LIN {X 0,Y 381.676,Z 552.93,A -85,B 0,C 180,E1 -11968.947,E2 -11968.947} C_VEL
LIN {X 0,Y 381.658,Z 553.223,A -85,B 0,C 180,E1 -11970.002,E2 -11970.002} C_VEL
LIN {X 0,Y 381.677,Z 553.115,A -85,B 0,C 180,E1 -11971.057,E2 -11971.057} C_VEL
LIN {X 0,Y 381.64,Z 552.556,A -85,B 0,C 180,E1 -11972.113,E2 -11972.113} C_VEL
LIN {X 0,Y 381.647,Z 550.205,A -85,B 0,C 180,E1 -11974.226,E2 -11974.226} C_VEL
LIN {X 0,Y 381.694,Z 546.609,A -85,B 0,C 180,E1 -11976.126,E2 -11976.126} C_VEL
LIN {X 0,Y 381.966,Z 541.741,A -85,B 0,C 180,E1 -11977.934,E2 -11977.934} C_VEL
LIN {X 0,Y 382.432,Z 535.151,A -85,B 0,C 180,E1 -11979.789,E2 -11979.789} C_VEL
LIN {X 0,Y 382.983,Z 527.932,A -85,B 0,C 180,E1 -11981.379,E2 -11981.379} C_VEL
LIN {X 0,Y 383.876,Z 518.998,A -85,B 0,C 180,E1 -11982.962,E2 -11982.962} C_VEL
LIN {X 0,Y 384.66,Z 509.425,A -85,B 0,C 180,E1 -11984.335,E2 -11984.335} C_VEL
LIN {X 0,Y 385.769,Z 498.433,A -85,B 0,C 180,E1 -11985.59,E2 -11985.59} C_VEL
LIN {X 0,Y 386.845,Z 487.015,A -85,B 0,C 180,E1 -11986.629,E2 -11986.629} C_VEL
LIN {X 0,Y 387.515,Z 477.015,A -85,B 0,C 180,E1 -11987.357,E2 -11987.357} C_VEL
LIN {X 0,Y 386.584,Z 463.507,A -85,B 0,C 180,E1 -11988.193,E2 -11988.193} C_VEL
LIN {X 0,Y 384.34,Z 449.997,A -85,B 0,C 180,E1 -11988.878,E2 -11988.878} C_VEL
LIN {X 0,Y 382.993,Z 443.041,A -85,B 0,C 180,E1 -11989.168,E2 -11989.168} C_VEL
LIN {X 0,Y 383.721,Z 433.258,A -85,B 0,C 180,E1 -11992.622,E2 -11992.622} C_VEL
LIN {X 0,Y 384.612,Z 423.855,A -85,B 0,C 180,E1 -11996.013,E2 -11996.013} C_VEL
LIN {X 0,Y 385.69,Z 414.532,A -85,B 0,C 180,E1 -11999.473,E2 -11999.473} C_VEL
LIN {X 0,Y 386.129,Z 410.031,A -85,B 0,C 180,E1 -12001.189,E2 -12001.189} C_VEL
LIN {X 0,Y 385.15,Z 403.611,A -85,B 0,C 180,E1 -12003.819,E2 -12003.819} C_VEL
LIN {X 0,Y 383.607,Z 395.835,A -85,B 0,C 180,E1 -12007.201,E2 -12007.201} C_VEL
LIN {X 0,Y 383.015,Z 392.777,A -85,B 0,C 180,E1 -12008.601,E2 -12008.601} C_VEL
LIN {X 0,Y 382.967,Z 392.783,A -85,B 0,C 180,E1 -12011.351,E2 -12011.351} C_VEL
LIN {X 0,Y 382.995,Z 392.777,A -85,B 0,C 180,E1 -12014.303,E2 -12014.303} C_VEL
LIN {X 0,Y 383.004,Z 392.776,A -85,B 0,C 180,E1 -12017.239,E2 -12017.239} C_VEL
LIN {X 0,Y 382.993,Z 392.777,A -85,B 0,C 180,E1 -12020.42,E2 -12020.42} C_VEL
LIN {X 0,Y 383.03,Z 392.774,A -85,B 0,C 180,E1 -12024.045,E2 -12024.045} C_VEL
LIN {X 0,Y 382.992,Z 392.778,A -85,B 0,C 180,E1 -12027.579,E2 -12027.579} C_VEL
LIN {X 0,Y 382.982,Z 392.779,A -85,B 0,C 180,E1 -12030.299,E2 -12030.299} C_VEL
LIN {X 0,Y 383.009,Z 392.775,A -85,B 0,C 180,E1 -12034.045,E2 -12034.045} C_VEL
LIN {X 0,Y 382.993,Z 392.778,A -85,B 0,C 180,E1 -12037.334,E2 -12037.334} C_VEL
LIN {X 0,Y 383.067,Z 392.771,A -85,B 0,C 180,E1 -12040.716,E2 -12040.716} C_VEL
LIN {X 0,Y 383.087,Z 392.771,A -85,B 0,C 180,E1 -12044.027,E2 -12044.027} C_VEL
LIN {X 0,Y 383.142,Z 392.763,A -85,B 0,C 180,E1 -12047.284,E2 -12047.284} C_VEL
LIN {X 0,Y 383.144,Z 392.76,A -85,B 0,C 180,E1 -12050.497,E2 -12050.497} C_VEL
LIN {X 0,Y 383.239,Z 392.75,A -85,B 0,C 180,E1 -12053.683,E2 -12053.683} C_VEL
LIN {X 0,Y 383.256,Z 392.948,A -85,B 0,C 180,E1 -12054.343,E2 -12054.343} C_VEL
LIN {X 0,Y 383.639,Z 397.881,A -85,B 0,C 180,E1 -12056.849,E2 -12056.849} C_VEL
LIN {X 0,Y 383.596,Z 403.09,A -85,B 0,C 180,E1 -12059.475,E2 -12059.475} C_VEL
LIN {X 0,Y 383.065,Z 411.611,A -85,B 0,C 180,E1 -12063.681,E2 -12063.681} C_VEL
LIN {X 0,Y 382.951,Z 417.902,A -85,B 0,C 180,E1 -12066.851,E2 -12066.851} C_VEL
LIN {X 0,Y 382.705,Z 424.252,A -85,B 0,C 180,E1 -12070.047,E2 -12070.047} C_VEL
LIN {X 0,Y 382.589,Z 427.474,A -85,B 0,C 180,E1 -12071.691,E2 -12071.691} C_VEL
LIN {X 0,Y 386.286,Z 441.807,A -85,B 0,C 180,E1 -12072.477,E2 -12072.477} C_VEL
LIN {X 0,Y 388.313,Z 452.899,A -85,B 0,C 180,E1 -12073.208,E2 -12073.208} C_VEL
LIN {X 0,Y 388.517,Z 456.626,A -85,B 0,C 180,E1 -12073.467,E2 -12073.467} C_VEL
LIN {X 0,Y 387.616,Z 468.027,A -85,B 0,C 180,E1 -12074.302,E2 -12074.302} C_VEL
LIN {X 0,Y 386.669,Z 479.198,A -85,B 0,C 180,E1 -12075.351,E2 -12075.351} C_VEL
LIN {X 0,Y 385.591,Z 490.485,A -85,B 0,C 180,E1 -12076.682,E2 -12076.682} C_VEL
LIN {X 0,Y 384.547,Z 500.254,A -85,B 0,C 180,E1 -12078.127,E2 -12078.127} C_VEL
LIN {X 0,Y 383.636,Z 509.359,A -85,B 0,C 180,E1 -12079.81,E2 -12079.81} C_VEL
LIN {X 0,Y 382.866,Z 516.695,A -85,B 0,C 180,E1 -12081.538,E2 -12081.538} C_VEL
LIN {X 0,Y 382.291,Z 522.218,A -85,B 0,C 180,E1 -12083.189,E2 -12083.189} C_VEL
LIN {X 0,Y 381.934,Z 526.91,A -85,B 0,C 180,E1 -12085.038,E2 -12085.038} C_VEL
LIN {X 0,Y 381.752,Z 529.124,A -85,B 0,C 180,E1 -12086.221,E2 -12086.221} C_VEL
LIN {X 0,Y 381.54,Z 531.322,A -85,B 0,C 180,E1 -12087.849,E2 -12087.849} C_VEL
LIN {X 0,Y 381.375,Z 532.743,A -85,B 0,C 180,E1 -12089.987,E2 -12089.987} C_VEL
LIN {X 0,Y 381.363,Z 532.498,A -85,B 0,C 180,E1 -12092.034,E2 -12092.034} C_VEL
LIN {X 0,Y 381.456,Z 530.872,A -85,B 0,C 180,E1 -12093.993,E2 -12093.993} C_VEL
LIN {X 0,Y 381.71,Z 527.886,A -85,B 0,C 180,E1 -12095.89,E2 -12095.89} C_VEL
LIN {X 0,Y 381.974,Z 523.67,A -85,B 0,C 180,E1 -12097.704,E2 -12097.704} C_VEL
LIN {X 0,Y 382.341,Z 518.193,A -85,B 0,C 180,E1 -12099.462,E2 -12099.462} C_VEL
LIN {X 0,Y 382.887,Z 511.233,A -85,B 0,C 180,E1 -12101.185,E2 -12101.185} C_VEL
LIN {X 0,Y 383.583,Z 502.634,A -85,B 0,C 180,E1 -12102.87,E2 -12102.87} C_VEL
LIN {X 0,Y 384.35,Z 493.592,A -85,B 0,C 180,E1 -12104.287,E2 -12104.287} C_VEL
LIN {X 0,Y 385.172,Z 483.42,A -85,B 0,C 180,E1 -12105.58,E2 -12105.58} C_VEL
LIN {X 0,Y 386.06,Z 472.137,A -85,B 0,C 180,E1 -12106.733,E2 -12106.733} C_VEL
LIN {X 0,Y 386.869,Z 460.044,A -85,B 0,C 180,E1 -12107.697,E2 -12107.697} C_VEL
LIN {X 0,Y 387.259,Z 452.848,A -85,B 0,C 180,E1 -12108.166,E2 -12108.166} C_VEL
LIN {X 0,Y 385.017,Z 440.265,A -85,B 0,C 180,E1 -12108.917,E2 -12108.917} C_VEL
LIN {X 0,Y 382.268,Z 426.607,A -85,B 0,C 180,E1 -12109.537,E2 -12109.537} C_VEL
LIN {X 0,Y 382.461,Z 419.18,A -85,B 0,C 180,E1 -12113.328,E2 -12113.328} C_VEL
LIN {X 0,Y 382.701,Z 412.84,A -85,B 0,C 180,E1 -12116.568,E2 -12116.568} C_VEL
LIN {X 0,Y 382.851,Z 406.873,A -85,B 0,C 180,E1 -12119.629,E2 -12119.629} C_VEL
LIN {X 0,Y 383.057,Z 399.753,A -85,B 0,C 180,E1 -12123.286,E2 -12123.286} C_VEL
LIN {X 0,Y 383.274,Z 394.063,A -85,B 0,C 180,E1 -12126.207,E2 -12126.207} C_VEL
LIN {X 0,Y 383.134,Z 392.763,A -85,B 0,C 180,E1 -12126.907,E2 -12126.907} C_VEL
LIN {X 0,Y 383.062,Z 392.772,A -85,B 0,C 180,E1 -12130.714,E2 -12130.714} C_VEL
LIN {X 0,Y 383.083,Z 392.767,A -85,B 0,C 180,E1 -12134.025,E2 -12134.025} C_VEL
LIN {X 0,Y 383.138,Z 392.76,A -85,B 0,C 180,E1 -12137.282,E2 -12137.282} C_VEL
LIN {X 0,Y 383.151,Z 392.758,A -85,B 0,C 180,E1 -12140.496,E2 -12140.496} C_VEL
LIN {X 0,Y 383.255,Z 392.748,A -85,B 0,C 180,E1 -12143.681,E2 -12143.681} C_VEL
LIN {X 0,Y 383.402,Z 392.882,A -85,B 0,C 180,E1 -12148.422,E2 -12148.422} C_VEL
LIN {X 0,Y 383.672,Z 395.201,A -85,B 0,C 180,E1 -12149.998,E2 -12149.998} C_VEL
LIN {X 0,Y 383.201,Z 400.099,A -85,B 0,C 180,E1 -12153.152,E2 -12153.152} C_VEL
LIN {X 0,Y 383.03,Z 405.091,A -85,B 0,C 180,E1 -12156.318,E2 -12156.318} C_VEL
LIN {X 0,Y 382.717,Z 410.229,A -85,B 0,C 180,E1 -12159.51,E2 -12159.51} C_VEL
LIN {X 0,Y 382.459,Z 416.09,A -85,B 0,C 180,E1 -12163.116,E2 -12163.116} C_VEL
LIN {X 0,Y 382.132,Z 422.772,A -85,B 0,C 180,E1 -12167.111,E2 -12167.111} C_VEL
LIN {X 0,Y 382.095,Z 423.941,A -85,B 0,C 180,E1 -12167.803,E2 -12167.803} C_VEL
LIN {X 0,Y 384.57,Z 436.385,A -85,B 0,C 180,E1 -12168.442,E2 -12168.442} C_VEL
LIN {X 0,Y 386.052,Z 446.599,A -85,B 0,C 180,E1 -12169.125,E2 -12169.125} C_VEL
LIN {X 0,Y 385.837,Z 451.459,A -85,B 0,C 180,E1 -12169.483,E2 -12169.483} C_VEL
LIN {X 0,Y 384.873,Z 456.639,A -85,B 0,C 180,E1 -12169.884,E2 -12169.884} C_VEL
LIN {X 0,Y 381.486,Z 464.749,A -85,B 0,C 180,E1 -12170.576,E2 -12170.576} C_VEL
LIN {X 0,Y 378.091,Z 472.32,A -85,B 0,C 180,E1 -12171.393,E2 -12171.393} C_VEL
LIN {X 0,Y 377.126,Z 476.647,A -85,B 0,C 180,E1 -12171.983,E2 -12171.983} C_VEL
LIN {X 0,Y 376.539,Z 483.312,A -85,B 0,C 180,E1 -12173.073,E2 -12173.073} C_VEL
LIN {X 0,Y 375.954,Z 490.705,A -85,B 0,C 180,E1 -12174.575,E2 -12174.575} C_VEL
LIN {X 0,Y 375.469,Z 496.349,A -85,B 0,C 180,E1 -12176.045,E2 -12176.045} C_VEL
LIN {X 0,Y 375.168,Z 500.199,A -85,B 0,C 180,E1 -12177.316,E2 -12177.316} C_VEL
LIN {X 0,Y 374.998,Z 502.515,A -85,B 0,C 180,E1 -12178.256,E2 -12178.256} C_VEL
LIN {X 0,Y 374.868,Z 504.313,A -85,B 0,C 180,E1 -12179.169,E2 -12179.169} C_VEL
LIN {X 0,Y 374.682,Z 506.2,A -85,B 0,C 180,E1 -12180.424,E2 -12180.424} C_VEL
LIN {X 0,Y 374.515,Z 507.759,A -85,B 0,C 180,E1 -12182.387,E2 -12182.387} C_VEL
LIN {X 0,Y 374.588,Z 507.67,A -85,B 0,C 180,E1 -12184.359,E2 -12184.359} C_VEL
LIN {X 0,Y 374.809,Z 506.038,A -85,B 0,C 180,E1 -12186.266,E2 -12186.266} C_VEL
LIN {X 0,Y 375.163,Z 502.8,A -85,B 0,C 180,E1 -12188.18,E2 -12188.18} C_VEL
LIN {X 0,Y 375.621,Z 498.336,A -85,B 0,C 180,E1 -12189.904,E2 -12189.904} C_VEL
LIN {X 0,Y 376.033,Z 493.712,A -85,B 0,C 180,E1 -12191.259,E2 -12191.259} C_VEL
LIN {X 0,Y 376.73,Z 486.408,A -85,B 0,C 180,E1 -12192.911,E2 -12192.911} C_VEL
LIN {X 0,Y 377.456,Z 478.658,A -85,B 0,C 180,E1 -12194.28,E2 -12194.28} C_VEL
LIN {X 0,Y 378.373,Z 469.354,A -85,B 0,C 180,E1 -12195.571,E2 -12195.571} C_VEL
LIN {X 0,Y 379.182,Z 459.767,A -85,B 0,C 180,E1 -12196.617,E2 -12196.617} C_VEL
LIN {X 0,Y 379.948,Z 448.957,A -85,B 0,C 180,E1 -12197.535,E2 -12197.535} C_VEL
LIN {X 0,Y 378.534,Z 439.629,A -85,B 0,C 180,E1 -12198.236,E2 -12198.236} C_VEL
LIN {X 0,Y 376.006,Z 428.04,A -85,B 0,C 180,E1 -12198.938,E2 -12198.938} C_VEL
LIN {X 0,Y 375.238,Z 424.84,A -85,B 0,C 180,E1 -12199.116,E2 -12199.116} C_VEL
LIN {X 0,Y 375.493,Z 419.416,A -85,B 0,C 180,E1 -12202.534,E2 -12202.534} C_VEL
LIN {X 0,Y 375.715,Z 414.233,A -85,B 0,C 180,E1 -12205.864,E2 -12205.864} C_VEL
LIN {X 0,Y 376.059,Z 408.313,A -85,B 0,C 180,E1 -12209.696,E2 -12209.696} C_VEL
LIN {X 0,Y 376.449,Z 402.826,A -85,B 0,C 180,E1 -12213.381,E2 -12213.381} C_VEL
LIN {X 0,Y 376.573,Z 398.851,A -85,B 0,C 180,E1 -12216.124,E2 -12216.124} C_VEL
LIN {X 0,Y 376.215,Z 394.642,A -85,B 0,C 180,E1 -12219.211,E2 -12219.211} C_VEL
LIN {X 0,Y 376.039,Z 393.648,A -85,B 0,C 180,E1 -12220.057,E2 -12220.057} C_VEL
LIN {X 0,Y 376.006,Z 393.654,A -85,B 0,C 180,E1 -12223.718,E2 -12223.718} C_VEL
LIN {X 0,Y 376.084,Z 393.64,A -85,B 0,C 180,E1 -12227.042,E2 -12227.042} C_VEL
LIN {X 0,Y 376.102,Z 393.638,A -85,B 0,C 180,E1 -12230.318,E2 -12230.318} C_VEL
LIN {X 0,Y 376.207,Z 393.625,A -85,B 0,C 180,E1 -12232.486,E2 -12232.486} C_VEL
LIN {X 0,Y 376.157,Z 393.631,A -85,B 0,C 180,E1 -12234.64,E2 -12234.64} C_VEL
LIN {X 0,Y 376.336,Z 393.608,A -85,B 0,C 180,E1 -12237.86,E2 -12237.86} C_VEL
LIN {X 0,Y 376.469,Z 393.592,A -85,B 0,C 180,E1 -12240,E2 -12240} C_VEL
LIN {X 0,Y 376.197,Z 393.624,A -85,B 0,C 180,E1 -12243.213,E2 -12243.213} C_VEL
LIN {X 0,Y 376.231,Z 393.616,A -85,B 0,C 180,E1 -12246.436,E2 -12246.436} C_VEL
LIN {X 0,Y 376.183,Z 393.627,A -85,B 0,C 180,E1 -12248.596,E2 -12248.596} C_VEL
LIN {X 0,Y 376.04,Z 393.643,A -85,B 0,C 180,E1 -12251.864,E2 -12251.864} C_VEL
LIN {X 0,Y 376.041,Z 393.642,A -85,B 0,C 180,E1 -12255.169,E2 -12255.169} C_VEL
LIN {X 0,Y 376.011,Z 393.643,A -85,B 0,C 180,E1 -12258.527,E2 -12258.527} C_VEL
LIN {X 0,Y 375.974,Z 393.65,A -85,B 0,C 180,E1 -12261.954,E2 -12261.954} C_VEL
LIN {X 0,Y 375.986,Z 393.651,A -85,B 0,C 180,E1 -12265.463,E2 -12265.463} C_VEL
LIN {X 0,Y 375.957,Z 393.653,A -85,B 0,C 180,E1 -12269.081,E2 -12269.081} C_VEL
LIN {X 0,Y 375.931,Z 393.655,A -85,B 0,C 180,E1 -12272.831,E2 -12272.831} C_VEL
LIN {X 0,Y 375.941,Z 393.657,A -85,B 0,C 180,E1 -12275.418,E2 -12275.418} C_VEL
LIN {X 0,Y 375.962,Z 393.656,A -85,B 0,C 180,E1 -12278.274,E2 -12278.274} C_VEL
LIN {X 0,Y 375.975,Z 393.654,A -85,B 0,C 180,E1 -12281.613,E2 -12281.613} C_VEL
LIN {X 0,Y 376.003,Z 393.647,A -85,B 0,C 180,E1 -12285.257,E2 -12285.257} C_VEL
LIN {X 0,Y 375.977,Z 393.652,A -85,B 0,C 180,E1 -12288.392,E2 -12288.392} C_VEL
LIN {X 0,Y 376.001,Z 393.84,A -85,B 0,C 180,E1 -12289.635,E2 -12289.635} C_VEL
LIN {X 0,Y 377.359,Z 400.688,A -85,B 0,C 180,E1 -12293.211,E2 -12293.211} C_VEL
LIN {X 0,Y 378.795,Z 407.795,A -85,B 0,C 180,E1 -12296.607,E2 -12296.607} C_VEL
LIN {X 0,Y 379.388,Z 412.708,A -85,B 0,C 180,E1 -12298.759,E2 -12298.759} C_VEL
LIN {X 0,Y 378.603,Z 418.588,A -85,B 0,C 180,E1 -12301.146,E2 -12301.146} C_VEL
LIN {X 0,Y 377.533,Z 427.623,A -85,B 0,C 180,E1 -12304.653,E2 -12304.653} C_VEL
LIN {X 0,Y 376.448,Z 438.252,A -85,B 0,C 180,E1 -12308.618,E2 -12308.618} C_VEL
LIN {X 0,Y 375.925,Z 445.155,A -85,B 0,C 180,E1 -12311.116,E2 -12311.116} C_VEL
LIN {X 0,Y 378.133,Z 458.373,A -85,B 0,C 180,E1 -12311.654,E2 -12311.654} C_VEL
LIN {X 0,Y 379.475,Z 470.242,A -85,B 0,C 180,E1 -12312.308,E2 -12312.308} C_VEL
LIN {X 0,Y 379.842,Z 479.385,A -85,B 0,C 180,E1 -12312.922,E2 -12312.922} C_VEL
LIN {X 0,Y 378.864,Z 490.974,A -85,B 0,C 180,E1 -12313.847,E2 -12313.847} C_VEL
LIN {X 0,Y 377.907,Z 501.428,A -85,B 0,C 180,E1 -12314.911,E2 -12314.911} C_VEL
LIN {X 0,Y 377.023,Z 511.942,A -85,B 0,C 180,E1 -12316.254,E2 -12316.254} C_VEL
LIN {X 0,Y 376.196,Z 521.916,A -85,B 0,C 180,E1 -12317.87,E2 -12317.87} C_VEL
LIN {X 0,Y 375.438,Z 530.272,A -85,B 0,C 180,E1 -12319.486,E2 -12319.486} C_VEL
LIN {X 0,Y 375.033,Z 537.056,A -85,B 0,C 180,E1 -12321.109,E2 -12321.109} C_VEL
LIN {X 0,Y 374.671,Z 543.237,A -85,B 0,C 180,E1 -12322.999,E2 -12322.999} C_VEL
LIN {X 0,Y 374.548,Z 547.21,A -85,B 0,C 180,E1 -12324.619,E2 -12324.619} C_VEL
LIN {X 0,Y 374.569,Z 549.239,A -85,B 0,C 180,E1 -12325.698,E2 -12325.698} C_VEL
LIN {X 0,Y 374.487,Z 550.836,A -85,B 0,C 180,E1 -12326.775,E2 -12326.775} C_VEL
LIN {X 0,Y 374.533,Z 552.006,A -85,B 0,C 180,E1 -12327.852,E2 -12327.852} C_VEL
LIN {X 0,Y 374.59,Z 552.716,A -85,B 0,C 180,E1 -12328.927,E2 -12328.927} C_VEL
LIN {X 0,Y 374.573,Z 553.022,A -85,B 0,C 180,E1 -12330.002,E2 -12330.002} C_VEL
LIN {X 0,Y 374.577,Z 552.929,A -85,B 0,C 180,E1 -12331.077,E2 -12331.077} C_VEL
LIN {X 0,Y 374.536,Z 552.395,A -85,B 0,C 180,E1 -12332.153,E2 -12332.153} C_VEL
LIN {X 0,Y 374.571,Z 550.068,A -85,B 0,C 180,E1 -12334.306,E2 -12334.306} C_VEL
LIN {X 0,Y 374.59,Z 546.878,A -85,B 0,C 180,E1 -12336.075,E2 -12336.075} C_VEL
LIN {X 0,Y 374.8,Z 543.253,A -85,B 0,C 180,E1 -12337.545,E2 -12337.545} C_VEL
LIN {X 0,Y 375.177,Z 538.17,A -85,B 0,C 180,E1 -12339.164,E2 -12339.164} C_VEL
LIN {X 0,Y 375.688,Z 531.777,A -85,B 0,C 180,E1 -12340.784,E2 -12340.784} C_VEL
LIN {X 0,Y 376.49,Z 523.791,A -85,B 0,C 180,E1 -12342.398,E2 -12342.398} C_VEL
LIN {X 0,Y 377.471,Z 513.894,A -85,B 0,C 180,E1 -12344.009,E2 -12344.009} C_VEL
LIN {X 0,Y 378.317,Z 504.705,A -85,B 0,C 180,E1 -12345.215,E2 -12345.215} C_VEL
LIN {X 0,Y 379.414,Z 493.4,A -85,B 0,C 180,E1 -12346.41,E2 -12346.41} C_VEL
LIN {X 0,Y 380.457,Z 482.611,A -85,B 0,C 180,E1 -12347.319,E2 -12347.319} C_VEL
LIN {X 0,Y 380.68,Z 475.754,A -85,B 0,C 180,E1 -12347.813,E2 -12347.813} C_VEL
LIN {X 0,Y 379.632,Z 462.562,A -85,B 0,C 180,E1 -12348.653,E2 -12348.653} C_VEL
LIN {X 0,Y 377.403,Z 449.462,A -85,B 0,C 180,E1 -12349.331,E2 -12349.331} C_VEL
LIN {X 0,Y 376.018,Z 442.443,A -85,B 0,C 180,E1 -12349.624,E2 -12349.624} C_VEL
LIN {X 0,Y 376.761,Z 432.936,A -85,B 0,C 180,E1 -12353.064,E2 -12353.064} C_VEL
LIN {X 0,Y 377.785,Z 422.997,A -85,B 0,C 180,E1 -12356.753,E2 -12356.753} C_VEL
LIN {X 0,Y 378.87,Z 414.284,A -85,B 0,C 180,E1 -12360.058,E2 -12360.058} C_VEL
LIN {X 0,Y 379.09,Z 410.668,A -85,B 0,C 180,E1 -12361.482,E2 -12361.482} C_VEL
LIN {X 0,Y 378.179,Z 404.934,A -85,B 0,C 180,E1 -12363.886,E2 -12363.886} C_VEL
LIN {X 0,Y 376.634,Z 397.166,A -85,B 0,C 180,E1 -12367.335,E2 -12367.335} C_VEL
LIN {X 0,Y 375.956,Z 393.656,A -85,B 0,C 180,E1 -12368.998,E2 -12368.998} C_VEL
LIN {X 0,Y 375.914,Z 393.661,A -85,B 0,C 180,E1 -12372.305,E2 -12372.305} C_VEL
LIN {X 0,Y 375.927,Z 393.658,A -85,B 0,C 180,E1 -12375.271,E2 -12375.271} C_VEL
LIN {X 0,Y 375.922,Z 393.657,A -85,B 0,C 180,E1 -12378.403,E2 -12378.403} C_VEL
LIN {X 0,Y 375.961,Z 393.647,A -85,B 0,C 180,E1 -12381.911,E2 -12381.911} C_VEL
LIN {X 0,Y 375.986,Z 393.65,A -85,B 0,C 180,E1 -12385.333,E2 -12385.333} C_VEL
LIN {X 0,Y 375.963,Z 393.653,A -85,B 0,C 180,E1 -12388.438,E2 -12388.438} C_VEL
LIN {X 0,Y 375.923,Z 393.659,A -85,B 0,C 180,E1 -12392.135,E2 -12392.135} C_VEL
LIN {X 0,Y 375.942,Z 393.657,A -85,B 0,C 180,E1 -12394.534,E2 -12394.534} C_VEL
LIN {X 0,Y 375.977,Z 393.654,A -85,B 0,C 180,E1 -12396.887,E2 -12396.887} C_VEL
LIN {X 0,Y 376.005,Z 393.65,A -85,B 0,C 180,E1 -12400.339,E2 -12400.339} C_VEL
LIN {X 0,Y 376.036,Z 393.647,A -85,B 0,C 180,E1 -12403.719,E2 -12403.719} C_VEL
LIN {X 0,Y 376.11,Z 393.639,A -85,B 0,C 180,E1 -12407.042,E2 -12407.042} C_VEL
LIN {X 0,Y 376.115,Z 393.636,A -85,B 0,C 180,E1 -12410.318,E2 -12410.318} C_VEL
LIN {X 0,Y 376.199,Z 393.628,A -85,B 0,C 180,E1 -12413.564,E2 -12413.564} C_VEL
LIN {X 0,Y 376.225,Z 393.864,A -85,B 0,C 180,E1 -12413.968,E2 -12413.968} C_VEL
LIN {X 0,Y 376.684,Z 398.262,A -85,B 0,C 180,E1 -12416.255,E2 -12416.255} C_VEL
LIN {X 0,Y 376.693,Z 403.468,A -85,B 0,C 180,E1 -12418.931,E2 -12418.931} C_VEL
LIN {X 0,Y 376.132,Z 410.892,A -85,B 0,C 180,E1 -12422.677,E2 -12422.677} C_VEL
LIN {X 0,Y 375.997,Z 417.246,A -85,B 0,C 180,E1 -12425.9,E2 -12425.9} C_VEL
LIN {X 0,Y 375.747,Z 423.599,A -85,B 0,C 180,E1 -12429.148,E2 -12429.148} C_VEL
LIN {X 0,Y 375.583,Z 427.665,A -85,B 0,C 180,E1 -12431.228,E2 -12431.228} C_VEL
LIN {X 0,Y 379.207,Z 441.095,A -85,B 0,C 180,E1 -12432,E2 -12432} C_VEL
LIN {X 0,Y 381.664,Z 454.259,A -85,B 0,C 180,E1 -12432.901,E2 -12432.901} C_VEL
LIN {X 0,Y 381.798,Z 457.974,A -85,B 0,C 180,E1 -12433.167,E2 -12433.167} C_VEL
LIN {X 0,Y 380.858,Z 469.124,A -85,B 0,C 180,E1 -12434.016,E2 -12434.016} C_VEL
LIN {X 0,Y 379.803,Z 480.885,A -85,B 0,C 180,E1 -12435.169,E2 -12435.169} C_VEL
LIN {X 0,Y 378.73,Z 491.28,A -85,B 0,C 180,E1 -12436.438,E2 -12436.438} C_VEL
LIN {X 0,Y 377.707,Z 500.463,A -85,B 0,C 180,E1 -12437.833,E2 -12437.833} C_VEL
LIN {X 0,Y 376.792,Z 508.515,A -85,B 0,C 180,E1 -12439.334,E2 -12439.334} C_VEL
LIN {X 0,Y 376.075,Z 515.211,A -85,B 0,C 180,E1 -12440.868,E2 -12440.868} C_VEL
LIN {X 0,Y 375.469,Z 521.15,A -85,B 0,C 180,E1 -12442.564,E2 -12442.564} C_VEL
LIN {X 0,Y 374.985,Z 525.932,A -85,B 0,C 180,E1 -12444.351,E2 -12444.351} C_VEL
LIN {X 0,Y 374.734,Z 528.885,A -85,B 0,C 180,E1 -12445.81,E2 -12445.81} C_VEL
LIN {X 0,Y 374.592,Z 530.352,A -85,B 0,C 180,E1 -12446.761,E2 -12446.761} C_VEL
LIN {X 0,Y 374.413,Z 531.874,A -85,B 0,C 180,E1 -12448.086,E2 -12448.086} C_VEL
LIN {X 0,Y 374.309,Z 532.662,A -85,B 0,C 180,E1 -12449.22,E2 -12449.22} C_VEL
LIN {X 0,Y 374.282,Z 533.009,A -85,B 0,C 180,E1 -12450.463,E2 -12450.463} C_VEL
LIN {X 0,Y 374.285,Z 532.537,A -85,B 0,C 180,E1 -12452.329,E2 -12452.329} C_VEL
LIN {X 0,Y 374.378,Z 530.662,A -85,B 0,C 180,E1 -12454.309,E2 -12454.309} C_VEL
LIN {X 0,Y 374.685,Z 527.458,A -85,B 0,C 180,E1 -12456.237,E2 -12456.237} C_VEL
LIN {X 0,Y 374.989,Z 522.688,A -85,B 0,C 180,E1 -12458.205,E2 -12458.205} C_VEL
LIN {X 0,Y 375.369,Z 517.326,A -85,B 0,C 180,E1 -12459.856,E2 -12459.856} C_VEL
LIN {X 0,Y 375.962,Z 510.124,A -85,B 0,C 180,E1 -12461.603,E2 -12461.603} C_VEL
LIN {X 0,Y 376.618,Z 502.301,A -85,B 0,C 180,E1 -12463.127,E2 -12463.127} C_VEL
LIN {X 0,Y 377.496,Z 492.518,A -85,B 0,C 180,E1 -12464.652,E2 -12464.652} C_VEL
LIN {X 0,Y 378.432,Z 481.589,A -85,B 0,C 180,E1 -12466.024,E2 -12466.024} C_VEL
LIN {X 0,Y 379.313,Z 470.131,A -85,B 0,C 180,E1 -12467.159,E2 -12467.159} C_VEL
LIN {X 0,Y 380.069,Z 458.885,A -85,B 0,C 180,E1 -12468.043,E2 -12468.043} C_VEL
LIN {X 0,Y 380.32,Z 453.733,A -85,B 0,C 180,E1 -12468.382,E2 -12468.382} C_VEL
LIN {X 0,Y 378.055,Z 440.908,A -85,B 0,C 180,E1 -12469.174,E2 -12469.174} C_VEL
LIN {X 0,Y 375.243,Z 426.749,A -85,B 0,C 180,E1 -12469.839,E2 -12469.839} C_VEL
LIN {X 0,Y 375.427,Z 419.449,A -85,B 0,C 180,E1 -12473.606,E2 -12473.606} C_VEL
LIN {X 0,Y 375.652,Z 413.832,A -85,B 0,C 180,E1 -12476.5,E2 -12476.5} C_VEL
LIN {X 0,Y 375.84,Z 406.523,A -85,B 0,C 180,E1 -12480.293,E2 -12480.293} C_VEL
LIN {X 0,Y 376.056,Z 399.809,A -85,B 0,C 180,E1 -12483.773,E2 -12483.773} C_VEL
LIN {X 0,Y 376.267,Z 395.061,A -85,B 0,C 180,E1 -12486.238,E2 -12486.238} C_VEL
LIN {X 0,Y 376.075,Z 393.642,A -85,B 0,C 180,E1 -12487.037,E2 -12487.037} C_VEL
LIN {X 0,Y 376.001,Z 393.652,A -85,B 0,C 180,E1 -12490.337,E2 -12490.337} C_VEL
LIN {X 0,Y 376.031,Z 393.647,A -85,B 0,C 180,E1 -12493.717,E2 -12493.717} C_VEL
LIN {X 0,Y 376.105,Z 393.638,A -85,B 0,C 180,E1 -12497.04,E2 -12497.04} C_VEL
LIN {X 0,Y 376.119,Z 393.635,A -85,B 0,C 180,E1 -12500.316,E2 -12500.316} C_VEL
LIN {X 0,Y 376.213,Z 393.626,A -85,B 0,C 180,E1 -12503.562,E2 -12503.562} C_VEL
LIN {X 0,Y 376.379,Z 393.768,A -85,B 0,C 180,E1 -12508.259,E2 -12508.259} C_VEL
LIN {X 0,Y 376.648,Z 396.289,A -85,B 0,C 180,E1 -12509.998,E2 -12509.998} C_VEL
LIN {X 0,Y 376.151,Z 401.221,A -85,B 0,C 180,E1 -12513.211,E2 -12513.211} C_VEL
LIN {X 0,Y 375.992,Z 406.2,A -85,B 0,C 180,E1 -12516.437,E2 -12516.437} C_VEL
LIN {X 0,Y 375.638,Z 411.396,A -85,B 0,C 180,E1 -12519.691,E2 -12519.691} C_VEL
LIN {X 0,Y 375.384,Z 417.059,A -85,B 0,C 180,E1 -12523.209,E2 -12523.209} C_VEL
LIN {X 0,Y 375.07,Z 423.5,A -85,B 0,C 180,E1 -12527.133,E2 -12527.133} C_VEL
LIN {X 0,Y 375.051,Z 424.132,A -85,B 0,C 180,E1 -12527.514,E2 -12527.514} C_VEL
LIN {X 0,Y 377.546,Z 436.626,A -85,B 0,C 180,E1 -12528.165,E2 -12528.165} C_VEL
LIN {X 0,Y 379.163,Z 447.635,A -85,B 0,C 180,E1 -12528.925,E2 -12528.925} C_VEL
LIN {X 0,Y 378.523,Z 458.305,A -85,B 0,C 180,E1 -12529.804,E2 -12529.804} C_VEL
LIN {X 0,Y 377.81,Z 466.882,A -85,B 0,C 180,E1 -12530.695,E2 -12530.695} C_VEL
LIN {X 0,Y 377.175,Z 475.938,A -85,B 0,C 180,E1 -12531.877,E2 -12531.877} C_VEL
LIN {X 0,Y 377.126,Z 476.647,A -85,B 0,C 180,E1 -12531.983,E2 -12531.983} C_VEL
LIN {X 0,Y 376.174,Z 480.782,A -85,B 0,C 180,E1 -12532.612,E2 -12532.612} C_VEL
LIN {X 0,Y 372.813,Z 487.054,A -85,B 0,C 180,E1 -12533.67,E2 -12533.67} C_VEL
LIN {X 0,Y 369.463,Z 492.64,A -85,B 0,C 180,E1 -12534.828,E2 -12534.828} C_VEL
LIN {X 0,Y 368.541,Z 495.629,A -85,B 0,C 180,E1 -12535.605,E2 -12535.605} C_VEL
LIN {X 0,Y 368.091,Z 500.708,A -85,B 0,C 180,E1 -12537.27,E2 -12537.27} C_VEL
LIN {X 0,Y 367.797,Z 504.779,A -85,B 0,C 180,E1 -12539.157,E2 -12539.157} C_VEL
LIN {X 0,Y 367.512,Z 507.327,A -85,B 0,C 180,E1 -12541.082,E2 -12541.082} C_VEL
LIN {X 0,Y 367.442,Z 508.246,A -85,B 0,C 180,E1 -12542.693,E2 -12542.693} C_VEL
LIN {X 0,Y 367.536,Z 507.958,A -85,B 0,C 180,E1 -12544.691,E2 -12544.691} C_VEL
LIN {X 0,Y 367.788,Z 506.1,A -85,B 0,C 180,E1 -12546.624,E2 -12546.624} C_VEL
LIN {X 0,Y 368.152,Z 502.798,A -85,B 0,C 180,E1 -12548.493,E2 -12548.493} C_VEL
LIN {X 0,Y 368.655,Z 498.031,A -85,B 0,C 180,E1 -12550.311,E2 -12550.311} C_VEL
LIN {X 0,Y 369.335,Z 491.593,A -85,B 0,C 180,E1 -12552.088,E2 -12552.088} C_VEL
LIN {X 0,Y 369.953,Z 485.03,A -85,B 0,C 180,E1 -12553.491,E2 -12553.491} C_VEL
LIN {X 0,Y 370.808,Z 476.694,A -85,B 0,C 180,E1 -12554.902,E2 -12554.902} C_VEL
LIN {X 0,Y 371.721,Z 467.566,A -85,B 0,C 180,E1 -12556.117,E2 -12556.117} C_VEL
LIN {X 0,Y 372.558,Z 457.945,A -85,B 0,C 180,E1 -12557.135,E2 -12557.135} C_VEL
LIN {X 0,Y 373.16,Z 449.897,A -85,B 0,C 180,E1 -12557.812,E2 -12557.812} C_VEL
LIN {X 0,Y 371.658,Z 440.355,A -85,B 0,C 180,E1 -12558.56,E2 -12558.56} C_VEL
LIN {X 0,Y 369.2,Z 429.165,A -85,B 0,C 180,E1 -12559.265,E2 -12559.265} C_VEL
LIN {X 0,Y 368.211,Z 425.112,A -85,B 0,C 180,E1 -12559.493,E2 -12559.493} C_VEL
LIN {X 0,Y 368.488,Z 419.297,A -85,B 0,C 180,E1 -12563.224,E2 -12563.224} C_VEL
LIN {X 0,Y 368.733,Z 414.351,A -85,B 0,C 180,E1 -12566.446,E2 -12566.446} C_VEL
LIN {X 0,Y 369.082,Z 408.516,A -85,B 0,C 180,E1 -12570.325,E2 -12570.325} C_VEL
LIN {X 0,Y 369.488,Z 403.046,A -85,B 0,C 180,E1 -12574.057,E2 -12574.057} C_VEL
LIN {X 0,Y 369.563,Z 399.679,A -85,B 0,C 180,E1 -12576.462,E2 -12576.462} C_VEL
LIN {X 0,Y 369.306,Z 396.544,A -85,B 0,C 180,E1 -12578.815,E2 -12578.815} C_VEL
LIN {X 0,Y 368.969,Z 394.531,A -85,B 0,C 180,E1 -12580.529,E2 -12580.529} C_VEL
LIN {X 0,Y 368.953,Z 394.533,A -85,B 0,C 180,E1 -12583.398,E2 -12583.398} C_VEL
LIN {X 0,Y 369.037,Z 394.518,A -85,B 0,C 180,E1 -12586.79,E2 -12586.79} C_VEL
LIN {X 0,Y 369.05,Z 394.516,A -85,B 0,C 180,E1 -12590.132,E2 -12590.132} C_VEL
LIN {X 0,Y 369.165,Z 394.501,A -85,B 0,C 180,E1 -12592.342,E2 -12592.342} C_VEL
LIN {X 0,Y 369.129,Z 394.507,A -85,B 0,C 180,E1 -12594.538,E2 -12594.538} C_VEL
LIN {X 0,Y 369.302,Z 394.484,A -85,B 0,C 180,E1 -12597.819,E2 -12597.819} C_VEL
LIN {X 0,Y 369.438,Z 394.467,A -85,B 0,C 180,E1 -12600,E2 -12600} C_VEL
LIN {X 0,Y 369.135,Z 394.502,A -85,B 0,C 180,E1 -12603.275,E2 -12603.275} C_VEL
LIN {X 0,Y 369.192,Z 394.492,A -85,B 0,C 180,E1 -12606.559,E2 -12606.559} C_VEL
LIN {X 0,Y 369.116,Z 394.506,A -85,B 0,C 180,E1 -12608.762,E2 -12608.762} C_VEL
LIN {X 0,Y 368.994,Z 394.52,A -85,B 0,C 180,E1 -12612.094,E2 -12612.094} C_VEL
LIN {X 0,Y 368.98,Z 394.52,A -85,B 0,C 180,E1 -12615.466,E2 -12615.466} C_VEL
LIN {X 0,Y 368.972,Z 394.521,A -85,B 0,C 180,E1 -12618.894,E2 -12618.894} C_VEL
LIN {X 0,Y 368.936,Z 394.53,A -85,B 0,C 180,E1 -12622.395,E2 -12622.395} C_VEL
LIN {X 0,Y 368.98,Z 394.525,A -85,B 0,C 180,E1 -12625.982,E2 -12625.982} C_VEL
LIN {X 0,Y 368.948,Z 394.527,A -85,B 0,C 180,E1 -12628.815,E2 -12628.815} C_VEL
LIN {X 0,Y 368.881,Z 394.532,A -85,B 0,C 180,E1 -12632.24,E2 -12632.24} C_VEL
LIN {X 0,Y 368.912,Z 394.533,A -85,B 0,C 180,E1 -12635.004,E2 -12635.004} C_VEL
LIN {X 0,Y 368.897,Z 394.535,A -85,B 0,C 180,E1 -12638.644,E2 -12638.644} C_VEL
LIN {X 0,Y 368.927,Z 394.532,A -85,B 0,C 180,E1 -12642.022,E2 -12642.022} C_VEL
LIN {X 0,Y 368.978,Z 394.522,A -85,B 0,C 180,E1 -12645.196,E2 -12645.196} C_VEL
LIN {X 0,Y 368.97,Z 394.618,A -85,B 0,C 180,E1 -12649.022,E2 -12649.022} C_VEL
LIN {X 0,Y 370.224,Z 401.253,A -85,B 0,C 180,E1 -12652.598,E2 -12652.598} C_VEL
LIN {X 0,Y 371.382,Z 406.9,A -85,B 0,C 180,E1 -12655.413,E2 -12655.413} C_VEL
LIN {X 0,Y 372.386,Z 412.74,A -85,B 0,C 180,E1 -12658.134,E2 -12658.134} C_VEL
LIN {X 0,Y 372.082,Z 417.043,A -85,B 0,C 180,E1 -12659.937,E2 -12659.937} C_VEL
LIN {X 0,Y 370.642,Z 427.518,A -85,B 0,C 180,E1 -12664.147,E2 -12664.147} C_VEL
LIN {X 0,Y 369.623,Z 436.652,A -85,B 0,C 180,E1 -12667.652,E2 -12667.652} C_VEL
LIN {X 0,Y 368.934,Z 444.899,A -85,B 0,C 180,E1 -12670.729,E2 -12670.729} C_VEL
LIN {X 0,Y 371.318,Z 458.654,A -85,B 0,C 180,E1 -12671.319,E2 -12671.319} C_VEL
LIN {X 0,Y 372.614,Z 470.677,A -85,B 0,C 180,E1 -12672.01,E2 -12672.01} C_VEL
LIN {X 0,Y 373.03,Z 479.154,A -85,B 0,C 180,E1 -12672.6,E2 -12672.6} C_VEL
LIN {X 0,Y 372.051,Z 490.701,A -85,B 0,C 180,E1 -12673.543,E2 -12673.543} C_VEL
LIN {X 0,Y 370.921,Z 502.191,A -85,B 0,C 180,E1 -12674.747,E2 -12674.747} C_VEL
LIN {X 0,Y 370.101,Z 511.625,A -85,B 0,C 180,E1 -12675.991,E2 -12675.991} C_VEL
LIN {X 0,Y 369.362,Z 520.08,A -85,B 0,C 180,E1 -12677.363,E2 -12677.363} C_VEL
LIN {X 0,Y 368.33,Z 531.08,A -85,B 0,C 180,E1 -12679.559,E2 -12679.559} C_VEL
LIN {X 0,Y 367.909,Z 537.685,A -85,B 0,C 180,E1 -12681.212,E2 -12681.212} C_VEL
LIN {X 0,Y 367.597,Z 542.904,A -85,B 0,C 180,E1 -12682.864,E2 -12682.864} C_VEL
LIN {X 0,Y 367.456,Z 546.917,A -85,B 0,C 180,E1 -12684.515,E2 -12684.515} C_VEL
LIN {X 0,Y 367.473,Z 548.964,A -85,B 0,C 180,E1 -12685.615,E2 -12685.615} C_VEL
LIN {X 0,Y 367.404,Z 550.577,A -85,B 0,C 180,E1 -12686.713,E2 -12686.713} C_VEL
LIN {X 0,Y 367.43,Z 551.772,A -85,B 0,C 180,E1 -12687.81,E2 -12687.81} C_VEL
LIN {X 0,Y 367.49,Z 552.501,A -85,B 0,C 180,E1 -12688.907,E2 -12688.907} C_VEL
LIN {X 0,Y 367.49,Z 552.821,A -85,B 0,C 180,E1 -12690.002,E2 -12690.002} C_VEL
LIN {X 0,Y 367.477,Z 552.742,A -85,B 0,C 180,E1 -12691.098,E2 -12691.098} C_VEL
LIN {X 0,Y 367.432,Z 552.237,A -85,B 0,C 180,E1 -12692.195,E2 -12692.195} C_VEL
LIN {X 0,Y 367.475,Z 549.944,A -85,B 0,C 180,E1 -12694.39,E2 -12694.39} C_VEL
LIN {X 0,Y 367.487,Z 547.127,A -85,B 0,C 180,E1 -12696.023,E2 -12696.023} C_VEL
LIN {X 0,Y 367.727,Z 543.2,A -85,B 0,C 180,E1 -12697.691,E2 -12697.691} C_VEL
LIN {X 0,Y 368.14,Z 538.152,A -85,B 0,C 180,E1 -12699.341,E2 -12699.341} C_VEL
LIN {X 0,Y 368.668,Z 531.81,A -85,B 0,C 180,E1 -12700.992,E2 -12700.992} C_VEL
LIN {X 0,Y 369.549,Z 523.879,A -85,B 0,C 180,E1 -12702.635,E2 -12702.635} C_VEL
LIN {X 0,Y 370.57,Z 514.072,A -85,B 0,C 180,E1 -12704.276,E2 -12704.276} C_VEL
LIN {X 0,Y 371.581,Z 503.883,A -85,B 0,C 180,E1 -12705.638,E2 -12705.638} C_VEL
LIN {X 0,Y 372.802,Z 492.51,A -85,B 0,C 180,E1 -12706.851,E2 -12706.851} C_VEL
LIN {X 0,Y 373.895,Z 481.624,A -85,B 0,C 180,E1 -12707.77,E2 -12707.77} C_VEL
LIN {X 0,Y 373.759,Z 471.947,A -85,B 0,C 180,E1 -12708.476,E2 -12708.476} C_VEL
LIN {X 0,Y 372.752,Z 461.71,A -85,B 0,C 180,E1 -12709.124,E2 -12709.124} C_VEL
LIN {X 0,Y 370.368,Z 448.324,A -85,B 0,C 180,E1 -12709.832,E2 -12709.832} C_VEL
LIN {X 0,Y 369.053,Z 441.811,A -85,B 0,C 180,E1 -12710.119,E2 -12710.119} C_VEL
LIN {X 0,Y 369.845,Z 432.645,A -85,B 0,C 180,E1 -12713.521,E2 -12713.521} C_VEL
LIN {X 0,Y 370.848,Z 423.335,A -85,B 0,C 180,E1 -12717.056,E2 -12717.056} C_VEL
LIN {X 0,Y 372.037,Z 414.023,A -85,B 0,C 180,E1 -12720.669,E2 -12720.669} C_VEL
LIN {X 0,Y 372.012,Z 410.925,A -85,B 0,C 180,E1 -12721.938,E2 -12721.938} C_VEL
LIN {X 0,Y 370.923,Z 404.685,A -85,B 0,C 180,E1 -12724.642,E2 -12724.642} C_VEL
LIN {X 0,Y 369.173,Z 395.863,A -85,B 0,C 180,E1 -12728.691,E2 -12728.691} C_VEL
LIN {X 0,Y 368.913,Z 394.534,A -85,B 0,C 180,E1 -12729.394,E2 -12729.394} C_VEL
LIN {X 0,Y 368.89,Z 394.536,A -85,B 0,C 180,E1 -12733.305,E2 -12733.305} C_VEL
LIN {X 0,Y 368.89,Z 394.529,A -85,B 0,C 180,E1 -12736.696,E2 -12736.696} C_VEL
LIN {X 0,Y 368.891,Z 394.531,A -85,B 0,C 180,E1 -12739.649,E2 -12739.649} C_VEL
LIN {X 0,Y 368.907,Z 394.532,A -85,B 0,C 180,E1 -12743.145,E2 -12743.145} C_VEL
LIN {X 0,Y 368.903,Z 394.534,A -85,B 0,C 180,E1 -12746.462,E2 -12746.462} C_VEL
LIN {X 0,Y 368.92,Z 394.529,A -85,B 0,C 180,E1 -12749.045,E2 -12749.045} C_VEL
LIN {X 0,Y 368.914,Z 394.533,A -85,B 0,C 180,E1 -12751.558,E2 -12751.558} C_VEL
LIN {X 0,Y 368.892,Z 394.537,A -85,B 0,C 180,E1 -12755.22,E2 -12755.22} C_VEL
LIN {X 0,Y 368.904,Z 394.533,A -85,B 0,C 180,E1 -12757.603,E2 -12757.603} C_VEL
LIN {X 0,Y 368.965,Z 394.526,A -85,B 0,C 180,E1 -12761.106,E2 -12761.106} C_VEL
LIN {X 0,Y 369.005,Z 394.524,A -85,B 0,C 180,E1 -12764.535,E2 -12764.535} C_VEL
LIN {X 0,Y 369.008,Z 394.521,A -85,B 0,C 180,E1 -12767.906,E2 -12767.906} C_VEL
LIN {X 0,Y 369.097,Z 394.511,A -85,B 0,C 180,E1 -12771.238,E2 -12771.238} C_VEL
LIN {X 0,Y 369.161,Z 394.591,A -85,B 0,C 180,E1 -12773.441,E2 -12773.441} C_VEL
LIN {X 0,Y 369.745,Z 399.693,A -85,B 0,C 180,E1 -12776.185,E2 -12776.185} C_VEL
LIN {X 0,Y 369.72,Z 404.867,A -85,B 0,C 180,E1 -12778.91,E2 -12778.91} C_VEL
LIN {X 0,Y 369.236,Z 411.341,A -85,B 0,C 180,E1 -12782.181,E2 -12782.181} C_VEL
LIN {X 0,Y 369.013,Z 417.686,A -85,B 0,C 180,E1 -12785.464,E2 -12785.464} C_VEL
LIN {X 0,Y 368.775,Z 424.05,A -85,B 0,C 180,E1 -12788.769,E2 -12788.769} C_VEL
LIN {X 0,Y 368.593,Z 427.855,A -85,B 0,C 180,E1 -12790.748,E2 -12790.748} C_VEL
LIN {X 0,Y 372.209,Z 440.893,A -85,B 0,C 180,E1 -12791.521,E2 -12791.521} C_VEL
LIN {X 0,Y 374.532,Z 452.337,A -85,B 0,C 180,E1 -12792.325,E2 -12792.325} C_VEL
LIN {X 0,Y 375.238,Z 457.698,A -85,B 0,C 180,E1 -12792.741,E2 -12792.741} C_VEL
LIN {X 0,Y 374.115,Z 470.203,A -85,B 0,C 180,E1 -12793.719,E2 -12793.719} C_VEL
LIN {X 0,Y 373.028,Z 481.613,A -85,B 0,C 180,E1 -12794.874,E2 -12794.874} C_VEL
LIN {X 0,Y 372.002,Z 490.433,A -85,B 0,C 180,E1 -12795.962,E2 -12795.962} C_VEL
LIN {X 0,Y 370.975,Z 499.719,A -85,B 0,C 180,E1 -12797.36,E2 -12797.36} C_VEL
LIN {X 0,Y 370.055,Z 507.674,A -85,B 0,C 180,E1 -12798.836,E2 -12798.836} C_VEL
LIN {X 0,Y 369.171,Z 515.079,A -85,B 0,C 180,E1 -12800.528,E2 -12800.528} C_VEL
LIN {X 0,Y 368.625,Z 519.707,A -85,B 0,C 180,E1 -12801.825,E2 -12801.825} C_VEL
LIN {X 0,Y 368.055,Z 524.89,A -85,B 0,C 180,E1 -12803.64,E2 -12803.64} C_VEL
LIN {X 0,Y 367.715,Z 528.709,A -85,B 0,C 180,E1 -12805.441,E2 -12805.441} C_VEL
LIN {X 0,Y 367.411,Z 531.425,A -85,B 0,C 180,E1 -12807.328,E2 -12807.328} C_VEL
LIN {X 0,Y 367.278,Z 532.525,A -85,B 0,C 180,E1 -12808.579,E2 -12808.579} C_VEL
LIN {X 0,Y 367.181,Z 533.221,A -85,B 0,C 180,E1 -12810.533,E2 -12810.533} C_VEL
LIN {X 0,Y 367.192,Z 532.508,A -85,B 0,C 180,E1 -12812.629,E2 -12812.629} C_VEL
LIN {X 0,Y 367.308,Z 530.423,A -85,B 0,C 180,E1 -12814.636,E2 -12814.636} C_VEL
LIN {X 0,Y 367.629,Z 527.037,A -85,B 0,C 180,E1 -12816.588,E2 -12816.588} C_VEL
LIN {X 0,Y 367.951,Z 522.383,A -85,B 0,C 180,E1 -12818.451,E2 -12818.451} C_VEL
LIN {X 0,Y 368.473,Z 515.815,A -85,B 0,C 180,E1 -12820.428,E2 -12820.428} C_VEL
LIN {X 0,Y 369.138,Z 507.835,A -85,B 0,C 180,E1 -12822.268,E2 -12822.268} C_VEL
LIN {X 0,Y 369.856,Z 499.704,A -85,B 0,C 180,E1 -12823.772,E2 -12823.772} C_VEL
LIN {X 0,Y 370.803,Z 489.756,A -85,B 0,C 180,E1 -12825.258,E2 -12825.258} C_VEL
LIN {X 0,Y 371.68,Z 479.272,A -85,B 0,C 180,E1 -12826.52,E2 -12826.52} C_VEL
LIN {X 0,Y 372.524,Z 468.447,A -85,B 0,C 180,E1 -12827.572,E2 -12827.572} C_VEL
LIN {X 0,Y 373.33,Z 457.297,A -85,B 0,C 180,E1 -12828.424,E2 -12828.424} C_VEL
LIN {X 0,Y 373.386,Z 454.491,A -85,B 0,C 180,E1 -12828.612,E2 -12828.612} C_VEL
LIN {X 0,Y 371.152,Z 441.72,A -85,B 0,C 180,E1 -12829.432,E2 -12829.432} C_VEL
LIN {X 0,Y 368.377,Z 428.145,A -85,B 0,C 180,E1 -12830.082,E2 -12830.082} C_VEL
LIN {X 0,Y 368.179,Z 426.883,A -85,B 0,C 180,E1 -12830.151,E2 -12830.151} C_VEL
LIN {X 0,Y 368.373,Z 419.994,A -85,B 0,C 180,E1 -12833.739,E2 -12833.739} C_VEL
LIN {X 0,Y 368.615,Z 413.696,A -85,B 0,C 180,E1 -12837.024,E2 -12837.024} C_VEL
LIN {X 0,Y 368.806,Z 407.444,A -85,B 0,C 180,E1 -12840.298,E2 -12840.298} C_VEL
LIN {X 0,Y 369.015,Z 401.294,A -85,B 0,C 180,E1 -12843.524,E2 -12843.524} C_VEL
LIN {X 0,Y 369.223,Z 395.749,A -85,B 0,C 180,E1 -12846.437,E2 -12846.437} C_VEL
LIN {X 0,Y 369.038,Z 394.519,A -85,B 0,C 180,E1 -12847.166,E2 -12847.166} C_VEL
LIN {X 0,Y 368.96,Z 394.526,A -85,B 0,C 180,E1 -12851.104,E2 -12851.104} C_VEL
LIN {X 0,Y 369,Z 394.52,A -85,B 0,C 180,E1 -12854.533,E2 -12854.533} C_VEL
LIN {X 0,Y 369.006,Z 394.521,A -85,B 0,C 180,E1 -12857.905,E2 -12857.905} C_VEL
LIN {X 0,Y 369.093,Z 394.512,A -85,B 0,C 180,E1 -12861.236,E2 -12861.236} C_VEL
LIN {X 0,Y 369.127,Z 394.509,A -85,B 0,C 180,E1 -12864.535,E2 -12864.535} C_VEL
LIN {X 0,Y 369.329,Z 394.648,A -85,B 0,C 180,E1 -12868.089,E2 -12868.089} C_VEL
LIN {X 0,Y 369.624,Z 397.392,A -85,B 0,C 180,E1 -12869.998,E2 -12869.998} C_VEL
LIN {X 0,Y 369.101,Z 402.34,A -85,B 0,C 180,E1 -12873.272,E2 -12873.272} C_VEL
LIN {X 0,Y 368.955,Z 407.344,A -85,B 0,C 180,E1 -12876.56,E2 -12876.56} C_VEL
LIN {X 0,Y 368.569,Z 412.556,A -85,B 0,C 180,E1 -12879.879,E2 -12879.879} C_VEL
LIN {X 0,Y 368.31,Z 417.994,A -85,B 0,C 180,E1 -12883.304,E2 -12883.304} C_VEL
LIN {X 0,Y 368.006,Z 424.344,A -85,B 0,C 180,E1 -12887.216,E2 -12887.216} C_VEL
LIN {X 0,Y 370.25,Z 435.563,A -85,B 0,C 180,E1 -12887.795,E2 -12887.795} C_VEL
LIN {X 0,Y 372.183,Z 447.363,A -85,B 0,C 180,E1 -12888.619,E2 -12888.619} C_VEL
LIN {X 0,Y 371.724,Z 457.146,A -85,B 0,C 180,E1 -12889.42,E2 -12889.42} C_VEL
LIN {X 0,Y 370.862,Z 467.64,A -85,B 0,C 180,E1 -12890.52,E2 -12890.52} C_VEL
LIN {X 0,Y 370.238,Z 476.098,A -85,B 0,C 180,E1 -12891.648,E2 -12891.648} C_VEL
LIN {X 0,Y 369.526,Z 483.936,A -85,B 0,C 180,E1 -12892.944,E2 -12892.944} C_VEL
LIN {X 0,Y 368.982,Z 490.599,A -85,B 0,C 180,E1 -12894.314,E2 -12894.314} C_VEL
LIN {X 0,Y 368.541,Z 495.629,A -85,B 0,C 180,E1 -12895.605,E2 -12895.605} C_VEL
LIN {X 0,Y 367.654,Z 498.36,A -85,B 0,C 180,E1 -12896.411,E2 -12896.411} C_VEL
LIN {X 0,Y 364.47,Z 502.205,A -85,B 0,C 180,E1 -12897.754,E2 -12897.754} C_VEL
LIN {X 0,Y 361.337,Z 505.263,A -85,B 0,C 180,E1 -12899.167,E2 -12899.167} C_VEL
LIN {X 0,Y 360.543,Z 506.555,A -85,B 0,C 180,E1 -12900.072,E2 -12900.072} C_VEL
LIN {X 0,Y 360.387,Z 508.258,A -85,B 0,C 180,E1 -12901.768,E2 -12901.768} C_VEL
LIN {X 0,Y 360.362,Z 508.723,A -85,B 0,C 180,E1 -12903.094,E2 -12903.094} C_VEL
LIN {X 0,Y 360.481,Z 508.183,A -85,B 0,C 180,E1 -12905.032,E2 -12905.032} C_VEL
LIN {X 0,Y 360.765,Z 506.162,A -85,B 0,C 180,E1 -12906.993,E2 -12906.993} C_VEL
LIN {X 0,Y 361.193,Z 502.645,A -85,B 0,C 180,E1 -12908.895,E2 -12908.895} C_VEL
LIN {X 0,Y 361.61,Z 498.942,A -85,B 0,C 180,E1 -12910.32,E2 -12910.32} C_VEL
LIN {X 0,Y 362.179,Z 493.518,A -85,B 0,C 180,E1 -12911.923,E2 -12911.923} C_VEL
LIN {X 0,Y 362.871,Z 486.951,A -85,B 0,C 180,E1 -12913.432,E2 -12913.432} C_VEL
LIN {X 0,Y 363.745,Z 478.971,A -85,B 0,C 180,E1 -12914.879,E2 -12914.879} C_VEL
LIN {X 0,Y 364.733,Z 469.825,A -85,B 0,C 180,E1 -12916.186,E2 -12916.186} C_VEL
LIN {X 0,Y 365.619,Z 460.216,A -85,B 0,C 180,E1 -12917.265,E2 -12917.265} C_VEL
LIN {X 0,Y 366.301,Z 450.432,A -85,B 0,C 180,E1 -12918.136,E2 -12918.136} C_VEL
LIN {X 0,Y 364.467,Z 439.072,A -85,B 0,C 180,E1 -12919.034,E2 -12919.034} C_VEL
LIN {X 0,Y 361.779,Z 427.779,A -85,B 0,C 180,E1 -12919.755,E2 -12919.755} C_VEL
LIN {X 0,Y 361.222,Z 425.361,A -85,B 0,C 180,E1 -12919.906,E2 -12919.906} C_VEL
LIN {X 0,Y 361.427,Z 420.702,A -85,B 0,C 180,E1 -12922.93,E2 -12922.93} C_VEL
LIN {X 0,Y 361.729,Z 415.073,A -85,B 0,C 180,E1 -12926.655,E2 -12926.655} C_VEL
LIN {X 0,Y 361.991,Z 410.613,A -85,B 0,C 180,E1 -12929.683,E2 -12929.683} C_VEL
LIN {X 0,Y 362.447,Z 405.049,A -85,B 0,C 180,E1 -12933.514,E2 -12933.514} C_VEL
LIN {X 0,Y 362.611,Z 401.663,A -85,B 0,C 180,E1 -12935.983,E2 -12935.983} C_VEL
LIN {X 0,Y 362.387,Z 398.238,A -85,B 0,C 180,E1 -12938.564,E2 -12938.564} C_VEL
LIN {X 0,Y 361.924,Z 395.408,A -85,B 0,C 180,E1 -12940.872,E2 -12940.872} C_VEL
LIN {X 0,Y 361.923,Z 395.408,A -85,B 0,C 180,E1 -12944.226,E2 -12944.226} C_VEL
LIN {X 0,Y 361.977,Z 395.398,A -85,B 0,C 180,E1 -12946.527,E2 -12946.527} C_VEL
LIN {X 0,Y 362.014,Z 395.392,A -85,B 0,C 180,E1 -12949.938,E2 -12949.938} C_VEL
LIN {X 0,Y 362.128,Z 395.377,A -85,B 0,C 180,E1 -12952.192,E2 -12952.192} C_VEL
LIN {X 0,Y 362.102,Z 395.382,A -85,B 0,C 180,E1 -12954.431,E2 -12954.431} C_VEL
LIN {X 0,Y 362.267,Z 395.361,A -85,B 0,C 180,E1 -12957.777,E2 -12957.777} C_VEL
LIN {X 0,Y 362.408,Z 395.343,A -85,B 0,C 180,E1 -12960,E2 -12960} C_VEL
LIN {X 0,Y 362.267,Z 395.362,A -85,B 0,C 180,E1 -12962.224,E2 -12962.224} C_VEL
LIN {X 0,Y 362.154,Z 395.369,A -85,B 0,C 180,E1 -12966.687,E2 -12966.687} C_VEL
LIN {X 0,Y 362.053,Z 395.384,A -85,B 0,C 180,E1 -12968.934,E2 -12968.934} C_VEL
LIN {X 0,Y 361.947,Z 395.396,A -85,B 0,C 180,E1 -12972.333,E2 -12972.333} C_VEL
LIN {X 0,Y 361.942,Z 395.4,A -85,B 0,C 180,E1 -12974.622,E2 -12974.622} C_VEL
LIN {X 0,Y 361.94,Z 395.397,A -85,B 0,C 180,E1 -12978.101,E2 -12978.101} C_VEL
LIN {X 0,Y 361.896,Z 395.402,A -85,B 0,C 180,E1 -12981.653,E2 -12981.653} C_VEL
LIN {X 0,Y 361.909,Z 395.404,A -85,B 0,C 180,E1 -12985.292,E2 -12985.292} C_VEL
LIN {X 0,Y 361.903,Z 395.404,A -85,B 0,C 180,E1 -12987.78,E2 -12987.78} C_VEL
LIN {X 0,Y 361.829,Z 395.415,A -85,B 0,C 180,E1 -12991.288,E2 -12991.288} C_VEL
LIN {X 0,Y 361.837,Z 395.414,A -85,B 0,C 180,E1 -12994.283,E2 -12994.283} C_VEL
LIN {X 0,Y 361.849,Z 395.413,A -85,B 0,C 180,E1 -12997.226,E2 -12997.226} C_VEL
LIN {X 0,Y 361.89,Z 395.408,A -85,B 0,C 180,E1 -13000.771,E2 -13000.771} C_VEL
LIN {X 0,Y 361.92,Z 395.405,A -85,B 0,C 180,E1 -13004.353,E2 -13004.353} C_VEL
LIN {X 0,Y 361.88,Z 395.409,A -85,B 0,C 180,E1 -13007.561,E2 -13007.561} C_VEL
LIN {X 0,Y 361.925,Z 395.639,A -85,B 0,C 180,E1 -13008.502,E2 -13008.502} C_VEL
LIN {X 0,Y 363.047,Z 401.363,A -85,B 0,C 180,E1 -13011.727,E2 -13011.727} C_VEL
LIN {X 0,Y 364.449,Z 408.378,A -85,B 0,C 180,E1 -13015.333,E2 -13015.333} C_VEL
LIN {X 0,Y 365.357,Z 413.583,A -85,B 0,C 180,E1 -13017.821,E2 -13017.821} C_VEL
LIN {X 0,Y 365.267,Z 417.035,A -85,B 0,C 180,E1 -13019.348,E2 -13019.348} C_VEL
LIN {X 0,Y 363.783,Z 427.406,A -85,B 0,C 180,E1 -13023.622,E2 -13023.622} C_VEL
LIN {X 0,Y 362.71,Z 436.5,A -85,B 0,C 180,E1 -13027.203,E2 -13027.203} C_VEL
LIN {X 0,Y 361.953,Z 444.623,A -85,B 0,C 180,E1 -13030.323,E2 -13030.323} C_VEL
LIN {X 0,Y 364.475,Z 459.018,A -85,B 0,C 180,E1 -13030.976,E2 -13030.976} C_VEL
LIN {X 0,Y 365.768,Z 470.992,A -85,B 0,C 180,E1 -13031.692,E2 -13031.692} C_VEL
LIN {X 0,Y 366.21,Z 478.974,A -85,B 0,C 180,E1 -13032.265,E2 -13032.265} C_VEL
LIN {X 0,Y 365.386,Z 489.043,A -85,B 0,C 180,E1 -13033.09,E2 -13033.09} C_VEL
LIN {X 0,Y 364.263,Z 499.708,A -85,B 0,C 180,E1 -13034.188,E2 -13034.188} C_VEL
LIN {X 0,Y 363.338,Z 509.411,A -85,B 0,C 180,E1 -13035.439,E2 -13035.439} C_VEL
LIN {X 0,Y 362.542,Z 518.224,A -85,B 0,C 180,E1 -13036.837,E2 -13036.837} C_VEL
LIN {X 0,Y 361.63,Z 526.755,A -85,B 0,C 180,E1 -13038.513,E2 -13038.513} C_VEL
LIN {X 0,Y 361.067,Z 534.121,A -85,B 0,C 180,E1 -13040.197,E2 -13040.197} C_VEL
LIN {X 0,Y 360.745,Z 539.149,A -85,B 0,C 180,E1 -13041.601,E2 -13041.601} C_VEL
LIN {X 0,Y 360.482,Z 543.996,A -85,B 0,C 180,E1 -13043.285,E2 -13043.285} C_VEL
LIN {X 0,Y 360.351,Z 547.679,A -85,B 0,C 180,E1 -13044.968,E2 -13044.968} C_VEL
LIN {X 0,Y 360.323,Z 550.303,A -85,B 0,C 180,E1 -13046.648,E2 -13046.648} C_VEL
LIN {X 0,Y 360.33,Z 551.52,A -85,B 0,C 180,E1 -13047.767,E2 -13047.767} C_VEL
LIN {X 0,Y 360.39,Z 552.28,A -85,B 0,C 180,E1 -13048.885,E2 -13048.885} C_VEL
LIN {X 0,Y 360.394,Z 552.618,A -85,B 0,C 180,E1 -13050.002,E2 -13050.002} C_VEL
LIN {X 0,Y 360.377,Z 552.556,A -85,B 0,C 180,E1 -13051.12,E2 -13051.12} C_VEL
LIN {X 0,Y 360.331,Z 552.083,A -85,B 0,C 180,E1 -13052.238,E2 -13052.238} C_VEL
LIN {X 0,Y 360.323,Z 551.156,A -85,B 0,C 180,E1 -13053.357,E2 -13053.357} C_VEL
LIN {X 0,Y 360.383,Z 549.824,A -85,B 0,C 180,E1 -13054.476,E2 -13054.476} C_VEL
LIN {X 0,Y 360.387,Z 547.372,A -85,B 0,C 180,E1 -13055.973,E2 -13055.973} C_VEL
LIN {X 0,Y 360.677,Z 543.146,A -85,B 0,C 180,E1 -13057.842,E2 -13057.842} C_VEL
LIN {X 0,Y 361.094,Z 538.134,A -85,B 0,C 180,E1 -13059.525,E2 -13059.525} C_VEL
LIN {X 0,Y 361.656,Z 531.859,A -85,B 0,C 180,E1 -13061.208,E2 -13061.208} C_VEL
LIN {X 0,Y 362.619,Z 524.034,A -85,B 0,C 180,E1 -13062.881,E2 -13062.881} C_VEL
LIN {X 0,Y 363.693,Z 514.312,A -85,B 0,C 180,E1 -13064.551,E2 -13064.551} C_VEL
LIN {X 0,Y 364.761,Z 504.259,A -85,B 0,C 180,E1 -13065.938,E2 -13065.938} C_VEL
LIN {X 0,Y 366.055,Z 493.008,A -85,B 0,C 180,E1 -13067.171,E2 -13067.171} C_VEL
LIN {X 0,Y 367.187,Z 482.202,A -85,B 0,C 180,E1 -13068.115,E2 -13068.115} C_VEL
LIN {X 0,Y 366.986,Z 471.694,A -85,B 0,C 180,E1 -13068.914,E2 -13068.914} C_VEL
LIN {X 0,Y 365.97,Z 461.631,A -85,B 0,C 180,E1 -13069.578,E2 -13069.578} C_VEL
LIN {X 0,Y 363.721,Z 448.794,A -85,B 0,C 180,E1 -13070.291,E2 -13070.291} C_VEL
LIN {X 0,Y 362.119,Z 441.048,A -85,B 0,C 180,E1 -13070.672,E2 -13070.672} C_VEL
LIN {X 0,Y 363.052,Z 430.985,A -85,B 0,C 180,E1 -13074.517,E2 -13074.517} C_VEL
LIN {X 0,Y 364.201,Z 421.477,A -85,B 0,C 180,E1 -13078.217,E2 -13078.217} C_VEL
LIN {X 0,Y 365.037,Z 415.297,A -85,B 0,C 180,E1 -13080.679,E2 -13080.679} C_VEL
LIN {X 0,Y 365.015,Z 411.923,A -85,B 0,C 180,E1 -13082.094,E2 -13082.094} C_VEL
LIN {X 0,Y 363.963,Z 405.969,A -85,B 0,C 180,E1 -13084.727,E2 -13084.727} C_VEL
LIN {X 0,Y 362.415,Z 398.2,A -85,B 0,C 180,E1 -13088.358,E2 -13088.358} C_VEL
LIN {X 0,Y 361.868,Z 395.411,A -85,B 0,C 180,E1 -13089.749,E2 -13089.749} C_VEL
LIN {X 0,Y 361.836,Z 395.414,A -85,B 0,C 180,E1 -13092.831,E2 -13092.831} C_VEL
LIN {X 0,Y 361.82,Z 395.409,A -85,B 0,C 180,E1 -13095.948,E2 -13095.948} C_VEL
LIN {X 0,Y 361.818,Z 395.41,A -85,B 0,C 180,E1 -13099.25,E2 -13099.25} C_VEL
LIN {X 0,Y 361.872,Z 395.408,A -85,B 0,C 180,E1 -13102.982,E2 -13102.982} C_VEL
LIN {X 0,Y 361.866,Z 395.41,A -85,B 0,C 180,E1 -13106.631,E2 -13106.631} C_VEL
LIN {X 0,Y 361.863,Z 395.413,A -85,B 0,C 180,E1 -13109.671,E2 -13109.671} C_VEL
LIN {X 0,Y 361.861,Z 395.411,A -85,B 0,C 180,E1 -13113.467,E2 -13113.467} C_VEL
LIN {X 0,Y 361.869,Z 395.41,A -85,B 0,C 180,E1 -13117.143,E2 -13117.143} C_VEL
LIN {X 0,Y 361.912,Z 395.406,A -85,B 0,C 180,E1 -13120.723,E2 -13120.723} C_VEL
LIN {X 0,Y 361.94,Z 395.402,A -85,B 0,C 180,E1 -13123.066,E2 -13123.066} C_VEL
LIN {X 0,Y 362.006,Z 395.395,A -85,B 0,C 180,E1 -13126.528,E2 -13126.528} C_VEL
LIN {X 0,Y 362.003,Z 395.395,A -85,B 0,C 180,E1 -13129.937,E2 -13129.937} C_VEL
LIN {X 0,Y 362.109,Z 395.496,A -85,B 0,C 180,E1 -13132.962,E2 -13132.962} C_VEL
LIN {X 0,Y 362.757,Z 400.161,A -85,B 0,C 180,E1 -13135.555,E2 -13135.555} C_VEL
LIN {X 0,Y 362.847,Z 405.383,A -85,B 0,C 180,E1 -13138.335,E2 -13138.335} C_VEL
LIN {X 0,Y 362.415,Z 410.664,A -85,B 0,C 180,E1 -13141.111,E2 -13141.111} C_VEL
LIN {X 0,Y 362.097,Z 418.13,A -85,B 0,C 180,E1 -13145.01,E2 -13145.01} C_VEL
LIN {X 0,Y 361.865,Z 423.609,A -85,B 0,C 180,E1 -13147.896,E2 -13147.896} C_VEL
LIN {X 0,Y 361.649,Z 428.012,A -85,B 0,C 180,E1 -13150.214,E2 -13150.214} C_VEL
LIN {X 0,Y 365.586,Z 442.07,A -85,B 0,C 180,E1 -13151.118,E2 -13151.118} C_VEL
LIN {X 0,Y 367.972,Z 453.905,A -85,B 0,C 180,E1 -13151.987,E2 -13151.987} C_VEL
LIN {X 0,Y 368.539,Z 459.522,A -85,B 0,C 180,E1 -13152.435,E2 -13152.435} C_VEL
LIN {X 0,Y 367.393,Z 471.399,A -85,B 0,C 180,E1 -13153.411,E2 -13153.411} C_VEL
LIN {X 0,Y 366.244,Z 482.64,A -85,B 0,C 180,E1 -13154.587,E2 -13154.587} C_VEL
LIN {X 0,Y 365.055,Z 492.652,A -85,B 0,C 180,E1 -13155.893,E2 -13155.893} C_VEL
LIN {X 0,Y 363.88,Z 502.097,A -85,B 0,C 180,E1 -13157.419,E2 -13157.419} C_VEL
LIN {X 0,Y 362.984,Z 509.154,A -85,B 0,C 180,E1 -13158.808,E2 -13158.808} C_VEL
LIN {X 0,Y 362.139,Z 516,A -85,B 0,C 180,E1 -13160.446,E2 -13160.446} C_VEL
LIN {X 0,Y 361.42,Z 522.046,A -85,B 0,C 180,E1 -13162.283,E2 -13162.283} C_VEL
LIN {X 0,Y 360.889,Z 526.704,A -85,B 0,C 180,E1 -13164.139,E2 -13164.139} C_VEL
LIN {X 0,Y 360.48,Z 530.469,A -85,B 0,C 180,E1 -13166.253,E2 -13166.253} C_VEL
LIN {X 0,Y 360.267,Z 532.329,A -85,B 0,C 180,E1 -13167.916,E2 -13167.916} C_VEL
LIN {X 0,Y 360.123,Z 533.124,A -85,B 0,C 180,E1 -13169.201,E2 -13169.201} C_VEL
LIN {X 0,Y 360.085,Z 533.396,A -85,B 0,C 180,E1 -13170.818,E2 -13170.818} C_VEL
LIN {X 0,Y 360.098,Z 532.451,A -85,B 0,C 180,E1 -13172.939,E2 -13172.939} C_VEL
LIN {X 0,Y 360.249,Z 530.171,A -85,B 0,C 180,E1 -13174.976,E2 -13174.976} C_VEL
LIN {X 0,Y 360.599,Z 526.525,A -85,B 0,C 180,E1 -13176.955,E2 -13176.955} C_VEL
LIN {X 0,Y 360.943,Z 521.685,A -85,B 0,C 180,E1 -13178.842,E2 -13178.842} C_VEL
LIN {X 0,Y 361.469,Z 515.49,A -85,B 0,C 180,E1 -13180.686,E2 -13180.686} C_VEL
LIN {X 0,Y 362.141,Z 507.741,A -85,B 0,C 180,E1 -13182.483,E2 -13182.483} C_VEL
LIN {X 0,Y 362.888,Z 499.582,A -85,B 0,C 180,E1 -13184.01,E2 -13184.01} C_VEL
LIN {X 0,Y 363.81,Z 490.278,A -85,B 0,C 180,E1 -13185.425,E2 -13185.425} C_VEL
LIN {X 0,Y 364.741,Z 479.495,A -85,B 0,C 180,E1 -13186.752,E2 -13186.752} C_VEL
LIN {X 0,Y 365.71,Z 467.782,A -85,B 0,C 180,E1 -13187.9,E2 -13187.9} C_VEL
LIN {X 0,Y 366.434,Z 455.367,A -85,B 0,C 180,E1 -13188.843,E2 -13188.843} C_VEL
LIN {X 0,Y 364.419,Z 443.468,A -85,B 0,C 180,E1 -13189.644,E2 -13189.644} C_VEL
LIN {X 0,Y 361.798,Z 430.31,A -85,B 0,C 180,E1 -13190.311,E2 -13190.311} C_VEL
LIN {X 0,Y 361.124,Z 427.01,A -85,B 0,C 180,E1 -13190.476,E2 -13190.476} C_VEL
LIN {X 0,Y 361.376,Z 419.734,A -85,B 0,C 180,E1 -13194.305,E2 -13194.305} C_VEL
LIN {X 0,Y 361.611,Z 413.312,A -85,B 0,C 180,E1 -13197.69,E2 -13197.69} C_VEL
LIN {X 0,Y 361.827,Z 407.164,A -85,B 0,C 180,E1 -13200.947,E2 -13200.947} C_VEL
LIN {X 0,Y 362.095,Z 400.045,A -85,B 0,C 180,E1 -13204.72,E2 -13204.72} C_VEL
LIN {X 0,Y 362.167,Z 396.605,A -85,B 0,C 180,E1 -13206.557,E2 -13206.557} C_VEL
LIN {X 0,Y 361.987,Z 395.397,A -85,B 0,C 180,E1 -13207.3,E2 -13207.3} C_VEL
LIN {X 0,Y 361.909,Z 395.407,A -85,B 0,C 180,E1 -13210.721,E2 -13210.721} C_VEL
LIN {X 0,Y 361.935,Z 395.401,A -85,B 0,C 180,E1 -13213.064,E2 -13213.064} C_VEL
LIN {X 0,Y 362,Z 395.395,A -85,B 0,C 180,E1 -13216.526,E2 -13216.526} C_VEL
LIN {X 0,Y 362.032,Z 395.392,A -85,B 0,C 180,E1 -13219.936,E2 -13219.936} C_VEL
LIN {X 0,Y 362.135,Z 395.38,A -85,B 0,C 180,E1 -13223.311,E2 -13223.311} C_VEL
LIN {X 0,Y 362.282,Z 395.528,A -85,B 0,C 180,E1 -13227.913,E2 -13227.913} C_VEL
LIN {X 0,Y 362.601,Z 398.5,A -85,B 0,C 180,E1 -13229.998,E2 -13229.998} C_VEL
LIN {X 0,Y 362.051,Z 403.451,A -85,B 0,C 180,E1 -13233.336,E2 -13233.336} C_VEL
LIN {X 0,Y 361.894,Z 408.511,A -85,B 0,C 180,E1 -13236.689,E2 -13236.689} C_VEL
LIN {X 0,Y 361.514,Z 413.715,A -85,B 0,C 180,E1 -13240.074,E2 -13240.074} C_VEL
LIN {X 0,Y 361.206,Z 419.113,A -85,B 0,C 180,E1 -13243.499,E2 -13243.499} C_VEL
LIN {X 0,Y 360.958,Z 424.574,A -85,B 0,C 180,E1 -13246.905,E2 -13246.905} C_VEL
LIN {X 0,Y 363.425,Z 436.856,A -85,B 0,C 180,E1 -13247.567,E2 -13247.567} C_VEL
LIN {X 0,Y 365.258,Z 448.228,A -85,B 0,C 180,E1 -13248.389,E2 -13248.389} C_VEL
LIN {X 0,Y 364.77,Z 458.344,A -85,B 0,C 180,E1 -13249.253,E2 -13249.253} C_VEL
LIN {X 0,Y 363.908,Z 468.394,A -85,B 0,C 180,E1 -13250.339,E2 -13250.339} C_VEL
LIN {X 0,Y 363.198,Z 477.274,A -85,B 0,C 180,E1 -13251.568,E2 -13251.568} C_VEL
LIN {X 0,Y 362.504,Z 484.56,A -85,B 0,C 180,E1 -13252.811,E2 -13252.811} C_VEL
LIN {X 0,Y 361.899,Z 491.698,A -85,B 0,C 180,E1 -13254.339,E2 -13254.339} C_VEL
LIN {X 0,Y 361.363,Z 497.416,A -85,B 0,C 180,E1 -13255.899,E2 -13255.899} C_VEL
LIN {X 0,Y 361.017,Z 501.213,A -85,B 0,C 180,E1 -13257.221,E2 -13257.221} C_VEL
LIN {X 0,Y 360.708,Z 505.248,A -85,B 0,C 180,E1 -13259.146,E2 -13259.146} C_VEL
LIN {X 0,Y 360.543,Z 506.555,A -85,B 0,C 180,E1 -13260.072,E2 -13260.072} C_VEL
LIN {X 0,Y 359.774,Z 507.693,A -85,B 0,C 180,E1 -13260.986,E2 -13260.986} C_VEL
LIN {X 0,Y 356.809,Z 508.802,A -85,B 0,C 180,E1 -13262.489,E2 -13262.489} C_VEL
LIN {X 0,Y 354.395,Z 509.053,A -85,B 0,C 180,E1 -13263.714,E2 -13263.714} C_VEL
LIN {X 0,Y 353.428,Z 508.844,A -85,B 0,C 180,E1 -13264.662,E2 -13264.662} C_VEL
LIN {X 0,Y 353.383,Z 508.62,A -85,B 0,C 180,E1 -13264.983,E2 -13264.983} C_VEL
LIN {X 0,Y 353.609,Z 507.224,A -85,B 0,C 180,E1 -13266.598,E2 -13266.598} C_VEL
LIN {X 0,Y 354.07,Z 503.919,A -85,B 0,C 180,E1 -13268.648,E2 -13268.648} C_VEL
LIN {X 0,Y 354.601,Z 499.454,A -85,B 0,C 180,E1 -13270.468,E2 -13270.468} C_VEL
LIN {X 0,Y 355.297,Z 493.463,A -85,B 0,C 180,E1 -13272.259,E2 -13272.259} C_VEL
LIN {X 0,Y 355.969,Z 487.238,A -85,B 0,C 180,E1 -13273.706,E2 -13273.706} C_VEL
LIN {X 0,Y 356.879,Z 479.443,A -85,B 0,C 180,E1 -13275.144,E2 -13275.144} C_VEL
LIN {X 0,Y 357.832,Z 470.9,A -85,B 0,C 180,E1 -13276.401,E2 -13276.401} C_VEL
LIN {X 0,Y 358.67,Z 462.236,A -85,B 0,C 180,E1 -13277.43,E2 -13277.43} C_VEL
LIN {X 0,Y 359.543,Z 452.394,A -85,B 0,C 180,E1 -13278.349,E2 -13278.349} C_VEL
LIN {X 0,Y 358.14,Z 442.615,A -85,B 0,C 180,E1 -13279.184,E2 -13279.184} C_VEL
LIN {X 0,Y 355.573,Z 431.159,A -85,B 0,C 180,E1 -13279.985,E2 -13279.985} C_VEL
LIN {X 0,Y 354.162,Z 425.632,A -85,B 0,C 180,E1 -13280.303,E2 -13280.303} C_VEL
LIN {X 0,Y 354.453,Z 420.805,A -85,B 0,C 180,E1 -13283.5,E2 -13283.5} C_VEL
LIN {X 0,Y 354.666,Z 416.604,A -85,B 0,C 180,E1 -13286.325,E2 -13286.325} C_VEL
LIN {X 0,Y 355.054,Z 410.801,A -85,B 0,C 180,E1 -13290.34,E2 -13290.34} C_VEL
LIN {X 0,Y 355.381,Z 407.111,A -85,B 0,C 180,E1 -13292.945,E2 -13292.945} C_VEL
LIN {X 0,Y 355.594,Z 403.678,A -85,B 0,C 180,E1 -13295.478,E2 -13295.478} C_VEL
LIN {X 0,Y 355.456,Z 399.924,A -85,B 0,C 180,E1 -13298.311,E2 -13298.311} C_VEL
LIN {X 0,Y 354.9,Z 396.284,A -85,B 0,C 180,E1 -13301.379,E2 -13301.379} C_VEL
LIN {X 0,Y 354.897,Z 396.282,A -85,B 0,C 180,E1 -13305.082,E2 -13305.082} C_VEL
LIN {X 0,Y 354.921,Z 396.275,A -85,B 0,C 180,E1 -13308.579,E2 -13308.579} C_VEL
LIN {X 0,Y 355.091,Z 396.253,A -85,B 0,C 180,E1 -13312.037,E2 -13312.037} C_VEL
LIN {X 0,Y 355.076,Z 396.256,A -85,B 0,C 180,E1 -13314.321,E2 -13314.321} C_VEL
LIN {X 0,Y 355.231,Z 396.238,A -85,B 0,C 180,E1 -13317.733,E2 -13317.733} C_VEL
LIN {X 0,Y 355.377,Z 396.219,A -85,B 0,C 180,E1 -13320,E2 -13320} C_VEL
LIN {X 0,Y 355.231,Z 396.238,A -85,B 0,C 180,E1 -13322.268,E2 -13322.268} C_VEL
LIN {X 0,Y 355.12,Z 396.245,A -85,B 0,C 180,E1 -13326.82,E2 -13326.82} C_VEL
LIN {X 0,Y 354.994,Z 396.263,A -85,B 0,C 180,E1 -13329.113,E2 -13329.113} C_VEL
LIN {X 0,Y 354.906,Z 396.273,A -85,B 0,C 180,E1 -13332.582,E2 -13332.582} C_VEL
LIN {X 0,Y 354.871,Z 396.278,A -85,B 0,C 180,E1 -13336.097,E2 -13336.097} C_VEL
LIN {X 0,Y 354.889,Z 396.274,A -85,B 0,C 180,E1 -13338.473,E2 -13338.473} C_VEL
LIN {X 0,Y 354.833,Z 396.284,A -85,B 0,C 180,E1 -13342.107,E2 -13342.107} C_VEL
LIN {X 0,Y 354.88,Z 396.281,A -85,B 0,C 180,E1 -13345.829,E2 -13345.829} C_VEL
LIN {X 0,Y 354.836,Z 396.281,A -85,B 0,C 180,E1 -13349.681,E2 -13349.681} C_VEL
LIN {X 0,Y 354.789,Z 396.292,A -85,B 0,C 180,E1 -13353.704,E2 -13353.704} C_VEL
LIN {X 0,Y 354.783,Z 396.293,A -85,B 0,C 180,E1 -13356.462,E2 -13356.462} C_VEL
LIN {X 0,Y 354.809,Z 396.291,A -85,B 0,C 180,E1 -13359.426,E2 -13359.426} C_VEL
LIN {X 0,Y 354.828,Z 396.288,A -85,B 0,C 180,E1 -13362.879,E2 -13362.879} C_VEL
LIN {X 0,Y 354.855,Z 396.285,A -85,B 0,C 180,E1 -13366.122,E2 -13366.122} C_VEL
LIN {X 0,Y 354.855,Z 396.456,A -85,B 0,C 180,E1 -13367.826,E2 -13367.826} C_VEL
LIN {X 0,Y 355.88,Z 401.503,A -85,B 0,C 180,E1 -13370.811,E2 -13370.811} C_VEL
LIN {X 0,Y 357.25,Z 408.459,A -85,B 0,C 180,E1 -13374.541,E2 -13374.541} C_VEL
LIN {X 0,Y 358.339,Z 414.45,A -85,B 0,C 180,E1 -13377.496,E2 -13377.496} C_VEL
LIN {X 0,Y 358.48,Z 417.062,A -85,B 0,C 180,E1 -13378.703,E2 -13378.703} C_VEL
LIN {X 0,Y 357.322,Z 424.353,A -85,B 0,C 180,E1 -13381.836,E2 -13381.836} C_VEL
LIN {X 0,Y 356.16,Z 433.321,A -85,B 0,C 180,E1 -13385.523,E2 -13385.523} C_VEL
LIN {X 0,Y 355.012,Z 444.18,A -85,B 0,C 180,E1 -13389.828,E2 -13389.828} C_VEL
LIN {X 0,Y 354.992,Z 444.452,A -85,B 0,C 180,E1 -13389.921,E2 -13389.921} C_VEL
LIN {X 0,Y 357.439,Z 458.049,A -85,B 0,C 180,E1 -13390.542,E2 -13390.542} C_VEL
LIN {X 0,Y 358.811,Z 469.303,A -85,B 0,C 180,E1 -13391.224,E2 -13391.224} C_VEL
LIN {X 0,Y 359.342,Z 480.585,A -85,B 0,C 180,E1 -13392.062,E2 -13392.062} C_VEL
LIN {X 0,Y 358.28,Z 491.693,A -85,B 0,C 180,E1 -13393.038,E2 -13393.038} C_VEL
LIN {X 0,Y 357.146,Z 501.941,A -85,B 0,C 180,E1 -13394.173,E2 -13394.173} C_VEL
LIN {X 0,Y 356.261,Z 511.091,A -85,B 0,C 180,E1 -13395.437,E2 -13395.437} C_VEL
LIN {X 0,Y 355.446,Z 519.486,A -85,B 0,C 180,E1 -13396.86,E2 -13396.86} C_VEL
LIN {X 0,Y 354.488,Z 527.679,A -85,B 0,C 180,E1 -13398.568,E2 -13398.568} C_VEL
LIN {X 0,Y 353.854,Z 535.804,A -85,B 0,C 180,E1 -13400.572,E2 -13400.572} C_VEL
LIN {X 0,Y 353.459,Z 542.148,A -85,B 0,C 180,E1 -13402.577,E2 -13402.577} C_VEL
LIN {X 0,Y 353.281,Z 546.258,A -85,B 0,C 180,E1 -13404.294,E2 -13404.294} C_VEL
LIN {X 0,Y 353.288,Z 548.371,A -85,B 0,C 180,E1 -13405.439,E2 -13405.439} C_VEL
LIN {X 0,Y 353.243,Z 550.024,A -85,B 0,C 180,E1 -13406.581,E2 -13406.581} C_VEL
LIN {X 0,Y 353.233,Z 551.261,A -85,B 0,C 180,E1 -13407.722,E2 -13407.722} C_VEL
LIN {X 0,Y 353.29,Z 552.058,A -85,B 0,C 180,E1 -13408.863,E2 -13408.863} C_VEL
LIN {X 0,Y 353.297,Z 552.415,A -85,B 0,C 180,E1 -13410.003,E2 -13410.003} C_VEL
LIN {X 0,Y 353.276,Z 552.369,A -85,B 0,C 180,E1 -13411.142,E2 -13411.142} C_VEL
LIN {X 0,Y 353.235,Z 551.922,A -85,B 0,C 180,E1 -13412.283,E2 -13412.283} C_VEL
LIN {X 0,Y 353.244,Z 551.022,A -85,B 0,C 180,E1 -13413.424,E2 -13413.424} C_VEL
LIN {X 0,Y 353.294,Z 549.704,A -85,B 0,C 180,E1 -13414.566,E2 -13414.566} C_VEL
LIN {X 0,Y 353.299,Z 547.585,A -85,B 0,C 180,E1 -13415.939,E2 -13415.939} C_VEL
LIN {X 0,Y 353.621,Z 543.118,A -85,B 0,C 180,E1 -13417.999,E2 -13417.999} C_VEL
LIN {X 0,Y 354.056,Z 538.169,A -85,B 0,C 180,E1 -13419.716,E2 -13419.716} C_VEL
LIN {X 0,Y 354.661,Z 531.942,A -85,B 0,C 180,E1 -13421.432,E2 -13421.432} C_VEL
LIN {X 0,Y 355.7,Z 524.204,A -85,B 0,C 180,E1 -13423.136,E2 -13423.136} C_VEL
LIN {X 0,Y 356.814,Z 514.553,A -85,B 0,C 180,E1 -13424.838,E2 -13424.838} C_VEL
LIN {X 0,Y 357.968,Z 504.642,A -85,B 0,C 180,E1 -13426.249,E2 -13426.249} C_VEL
LIN {X 0,Y 359.316,Z 493.577,A -85,B 0,C 180,E1 -13427.503,E2 -13427.503} C_VEL
LIN {X 0,Y 360.655,Z 481.225,A -85,B 0,C 180,E1 -13428.61,E2 -13428.61} C_VEL
LIN {X 0,Y 360.112,Z 468.659,A -85,B 0,C 180,E1 -13429.573,E2 -13429.573} C_VEL
LIN {X 0,Y 358.228,Z 455.33,A -85,B 0,C 180,E1 -13430.437,E2 -13430.437} C_VEL
LIN {X 0,Y 355.158,Z 440.357,A -85,B 0,C 180,E1 -13431.227,E2 -13431.227} C_VEL
LIN {X 0,Y 356.184,Z 430.246,A -85,B 0,C 180,E1 -13435.181,E2 -13435.181} C_VEL
LIN {X 0,Y 357.343,Z 421.2,A -85,B 0,C 180,E1 -13438.808,E2 -13438.808} C_VEL
LIN {X 0,Y 358.156,Z 415.014,A -85,B 0,C 180,E1 -13441.334,E2 -13441.334} C_VEL
LIN {X 0,Y 357.559,Z 410.345,A -85,B 0,C 180,E1 -13443.393,E2 -13443.393} C_VEL
LIN {X 0,Y 356.328,Z 404.135,A -85,B 0,C 180,E1 -13446.28,E2 -13446.28} C_VEL
LIN {X 0,Y 354.82,Z 396.359,A -85,B 0,C 180,E1 -13450.089,E2 -13450.089} C_VEL
LIN {X 0,Y 354.769,Z 396.294,A -85,B 0,C 180,E1 -13453.898,E2 -13453.898} C_VEL
LIN {X 0,Y 354.792,Z 396.291,A -85,B 0,C 180,E1 -13457.662,E2 -13457.662} C_VEL
LIN {X 0,Y 354.793,Z 396.292,A -85,B 0,C 180,E1 -13460.663,E2 -13460.663} C_VEL
LIN {X 0,Y 354.829,Z 396.286,A -85,B 0,C 180,E1 -13464.302,E2 -13464.302} C_VEL
LIN {X 0,Y 354.794,Z 396.291,A -85,B 0,C 180,E1 -13467.667,E2 -13467.667} C_VEL
LIN {X 0,Y 354.796,Z 396.291,A -85,B 0,C 180,E1 -13471.614,E2 -13471.614} C_VEL
LIN {X 0,Y 354.811,Z 396.289,A -85,B 0,C 180,E1 -13475.42,E2 -13475.42} C_VEL
LIN {X 0,Y 354.833,Z 396.288,A -85,B 0,C 180,E1 -13479.113,E2 -13479.113} C_VEL
LIN {X 0,Y 354.906,Z 396.28,A -85,B 0,C 180,E1 -13482.72,E2 -13482.72} C_VEL
LIN {X 0,Y 354.959,Z 396.271,A -85,B 0,C 180,E1 -13486.255,E2 -13486.255} C_VEL
LIN {X 0,Y 354.96,Z 396.271,A -85,B 0,C 180,E1 -13489.735,E2 -13489.735} C_VEL
LIN {X 0,Y 355.079,Z 396.459,A -85,B 0,C 180,E1 -13492.465,E2 -13492.465} C_VEL
LIN {X 0,Y 355.767,Z 400.668,A -85,B 0,C 180,E1 -13494.9,E2 -13494.9} C_VEL
LIN {X 0,Y 355.916,Z 404.787,A -85,B 0,C 180,E1 -13497.17,E2 -13497.17} C_VEL
LIN {X 0,Y 355.779,Z 409.013,A -85,B 0,C 180,E1 -13499.434,E2 -13499.434} C_VEL
LIN {X 0,Y 355.177,Z 417.566,A -85,B 0,C 180,E1 -13503.971,E2 -13503.971} C_VEL
LIN {X 0,Y 354.902,Z 424.425,A -85,B 0,C 180,E1 -13507.647,E2 -13507.647} C_VEL
LIN {X 0,Y 354.724,Z 428.449,A -85,B 0,C 180,E1 -13509.695,E2 -13509.695} C_VEL
LIN {X 0,Y 358.79,Z 442.303,A -85,B 0,C 180,E1 -13510.617,E2 -13510.617} C_VEL
LIN {X 0,Y 361.131,Z 453.896,A -85,B 0,C 180,E1 -13511.506,E2 -13511.506} C_VEL
LIN {X 0,Y 361.937,Z 460.295,A -85,B 0,C 180,E1 -13512.048,E2 -13512.048} C_VEL
LIN {X 0,Y 360.732,Z 472.207,A -85,B 0,C 180,E1 -13513.056,E2 -13513.056} C_VEL
LIN {X 0,Y 359.483,Z 483.647,A -85,B 0,C 180,E1 -13514.289,E2 -13514.289} C_VEL
LIN {X 0,Y 358.16,Z 494.17,A -85,B 0,C 180,E1 -13515.721,E2 -13515.721} C_VEL
LIN {X 0,Y 357,Z 502.857,A -85,B 0,C 180,E1 -13517.175,E2 -13517.175} C_VEL
LIN {X 0,Y 356.035,Z 510.06,A -85,B 0,C 180,E1 -13518.644,E2 -13518.644} C_VEL
LIN {X 0,Y 355.027,Z 517.619,A -85,B 0,C 180,E1 -13520.571,E2 -13520.571} C_VEL
LIN {X 0,Y 354.394,Z 522.501,A -85,B 0,C 180,E1 -13522.135,E2 -13522.135} C_VEL
LIN {X 0,Y 353.833,Z 527.002,A -85,B 0,C 180,E1 -13523.979,E2 -13523.979} C_VEL
LIN {X 0,Y 353.453,Z 530.452,A -85,B 0,C 180,E1 -13525.941,E2 -13525.941} C_VEL
LIN {X 0,Y 353.229,Z 532.006,A -85,B 0,C 180,E1 -13527.233,E2 -13527.233} C_VEL
LIN {X 0,Y 353.06,Z 533.227,A -85,B 0,C 180,E1 -13528.85,E2 -13528.85} C_VEL
LIN {X 0,Y 352.999,Z 533.53,A -85,B 0,C 180,E1 -13531.115,E2 -13531.115} C_VEL
LIN {X 0,Y 353.005,Z 532.371,A -85,B 0,C 180,E1 -13533.258,E2 -13533.258} C_VEL
LIN {X 0,Y 353.218,Z 529.809,A -85,B 0,C 180,E1 -13535.333,E2 -13535.333} C_VEL
LIN {X 0,Y 353.587,Z 525.977,A -85,B 0,C 180,E1 -13537.338,E2 -13537.338} C_VEL
LIN {X 0,Y 354.005,Z 520.322,A -85,B 0,C 180,E1 -13539.441,E2 -13539.441} C_VEL
LIN {X 0,Y 354.591,Z 513.536,A -85,B 0,C 180,E1 -13541.355,E2 -13541.355} C_VEL
LIN {X 0,Y 355.246,Z 506.47,A -85,B 0,C 180,E1 -13542.945,E2 -13542.945} C_VEL
LIN {X 0,Y 356.092,Z 498.103,A -85,B 0,C 180,E1 -13544.471,E2 -13544.471} C_VEL
LIN {X 0,Y 357.044,Z 488.32,A -85,B 0,C 180,E1 -13545.927,E2 -13545.927} C_VEL
LIN {X 0,Y 357.997,Z 477.792,A -85,B 0,C 180,E1 -13547.199,E2 -13547.199} C_VEL
LIN {X 0,Y 358.953,Z 466.019,A -85,B 0,C 180,E1 -13548.323,E2 -13548.323} C_VEL
LIN {X 0,Y 359.478,Z 456.125,A -85,B 0,C 180,E1 -13549.083,E2 -13549.083} C_VEL
LIN {X 0,Y 357.269,Z 442.987,A -85,B 0,C 180,E1 -13549.982,E2 -13549.982} C_VEL
LIN {X 0,Y 354.465,Z 429.291,A -85,B 0,C 180,E1 -13550.679,E2 -13550.679} C_VEL
LIN {X 0,Y 354.074,Z 427.136,A -85,B 0,C 180,E1 -13550.811,E2 -13550.811} C_VEL
LIN {X 0,Y 354.339,Z 420.37,A -85,B 0,C 180,E1 -13554.409,E2 -13554.409} C_VEL
LIN {X 0,Y 354.559,Z 414.302,A -85,B 0,C 180,E1 -13557.641,E2 -13557.641} C_VEL
LIN {X 0,Y 354.77,Z 408.677,A -85,B 0,C 180,E1 -13560.649,E2 -13560.649} C_VEL
LIN {X 0,Y 354.998,Z 402.104,A -85,B 0,C 180,E1 -13564.178,E2 -13564.178} C_VEL
LIN {X 0,Y 355.117,Z 397.465,A -85,B 0,C 180,E1 -13566.681,E2 -13566.681} C_VEL
LIN {X 0,Y 354.936,Z 396.275,A -85,B 0,C 180,E1 -13567.439,E2 -13567.439} C_VEL
LIN {X 0,Y 354.925,Z 396.276,A -85,B 0,C 180,E1 -13571.89,E2 -13571.89} C_VEL
LIN {X 0,Y 354.944,Z 396.272,A -85,B 0,C 180,E1 -13575.979,E2 -13575.979} C_VEL
LIN {X 0,Y 354.978,Z 396.27,A -85,B 0,C 180,E1 -13579.734,E2 -13579.734} C_VEL
LIN {X 0,Y 355.1,Z 396.255,A -85,B 0,C 180,E1 -13583.178,E2 -13583.178} C_VEL
LIN {X 0,Y 355.228,Z 396.41,A -85,B 0,C 180,E1 -13587.73,E2 -13587.73} C_VEL
LIN {X 0,Y 355.576,Z 399.575,A -85,B 0,C 180,E1 -13589.997,E2 -13589.997} C_VEL
LIN {X 0,Y 355.002,Z 404.56,A -85,B 0,C 180,E1 -13593.402,E2 -13593.402} C_VEL
LIN {X 0,Y 354.834,Z 409.633,A -85,B 0,C 180,E1 -13596.822,E2 -13596.822} C_VEL
LIN {X 0,Y 354.431,Z 414.929,A -85,B 0,C 180,E1 -13600.277,E2 -13600.277} C_VEL
LIN {X 0,Y 354.098,Z 420.352,A -85,B 0,C 180,E1 -13603.776,E2 -13603.776} C_VEL
LIN {X 0,Y 353.93,Z 424.783,A -85,B 0,C 180,E1 -13606.582,E2 -13606.582} C_VEL
LIN {X 0,Y 356.429,Z 437.37,A -85,B 0,C 180,E1 -13607.281,E2 -13607.281} C_VEL
LIN {X 0,Y 358.311,Z 448.864,A -85,B 0,C 180,E1 -13608.138,E2 -13608.138} C_VEL
LIN {X 0,Y 357.955,Z 457.667,A -85,B 0,C 180,E1 -13608.899,E2 -13608.899} C_VEL
LIN {X 0,Y 357.041,Z 467.818,A -85,B 0,C 180,E1 -13609.996,E2 -13609.996} C_VEL
LIN {X 0,Y 356.3,Z 476.905,A -85,B 0,C 180,E1 -13611.247,E2 -13611.247} C_VEL
LIN {X 0,Y 355.482,Z 485.151,A -85,B 0,C 180,E1 -13612.673,E2 -13612.673} C_VEL
LIN {X 0,Y 354.83,Z 492.68,A -85,B 0,C 180,E1 -13614.342,E2 -13614.342} C_VEL
LIN {X 0,Y 354.282,Z 498.094,A -85,B 0,C 180,E1 -13615.872,E2 -13615.872} C_VEL
LIN {X 0,Y 353.96,Z 501.696,A -85,B 0,C 180,E1 -13617.169,E2 -13617.169} C_VEL
LIN {X 0,Y 353.66,Z 505.533,A -85,B 0,C 180,E1 -13619.029,E2 -13619.029} C_VEL
LIN {X 0,Y 353.36,Z 508.189,A -85,B 0,C 180,E1 -13621.135,E2 -13621.135} C_VEL
LIN {X 0,Y 353.269,Z 509,A -85,B 0,C 180,E1 -13622.485,E2 -13622.485} C_VEL
LIN {X 0,Y 353.308,Z 509.104,A -85,B 0,C 180,E1 -13623.843,E2 -13623.843} C_VEL
LIN {X 0,Y 353.383,Z 508.62,A -85,B 0,C 180,E1 -13624.983,E2 -13624.983} C_VEL
LIN {X 0,Y 352.848,Z 508.06,A -85,B 0,C 180,E1 -13625.934,E2 -13625.934} C_VEL
LIN {X 0,Y 350.245,Z 506.455,A -85,B 0,C 180,E1 -13627.474,E2 -13627.474} C_VEL
LIN {X 0,Y 347.729,Z 503.889,A -85,B 0,C 180,E1 -13629,E2 -13629} C_VEL
LIN {X 0,Y 347.342,Z 501.818,A -85,B 0,C 180,E1 -13629.915,E2 -13629.915} C_VEL
LIN {X 0,Y 347.938,Z 496.904,A -85,B 0,C 180,E1 -13631.638,E2 -13631.638} C_VEL
LIN {X 0,Y 348.813,Z 489.786,A -85,B 0,C 180,E1 -13633.504,E2 -13633.504} C_VEL
LIN {X 0,Y 349.718,Z 482.192,A -85,B 0,C 180,E1 -13635.033,E2 -13635.033} C_VEL
LIN {X 0,Y 350.721,Z 473.948,A -85,B 0,C 180,E1 -13636.36,E2 -13636.36} C_VEL
LIN {X 0,Y 351.805,Z 463.696,A -85,B 0,C 180,E1 -13637.654,E2 -13637.654} C_VEL
LIN {X 0,Y 352.779,Z 453.592,A -85,B 0,C 180,E1 -13638.642,E2 -13638.642} C_VEL
LIN {X 0,Y 351.237,Z 442.867,A -85,B 0,C 180,E1 -13639.589,E2 -13639.589} C_VEL
LIN {X 0,Y 348.654,Z 431.576,A -85,B 0,C 180,E1 -13640.404,E2 -13640.404} C_VEL
LIN {X 0,Y 347.158,Z 425.862,A -85,B 0,C 180,E1 -13640.761,E2 -13640.761} C_VEL
LIN {X 0,Y 347.456,Z 420.946,A -85,B 0,C 180,E1 -13644.086,E2 -13644.086} C_VEL
LIN {X 0,Y 347.68,Z 416.836,A -85,B 0,C 180,E1 -13646.923,E2 -13646.923} C_VEL
LIN {X 0,Y 348.126,Z 411.034,A -85,B 0,C 180,E1 -13651.02,E2 -13651.02} C_VEL
LIN {X 0,Y 348.445,Z 407.415,A -85,B 0,C 180,E1 -13653.658,E2 -13653.658} C_VEL
LIN {X 0,Y 348.584,Z 404.016,A -85,B 0,C 180,E1 -13656.22,E2 -13656.22} C_VEL
LIN {X 0,Y 348.408,Z 400.801,A -85,B 0,C 180,E1 -13658.71,E2 -13658.71} C_VEL
LIN {X 0,Y 347.855,Z 397.162,A -85,B 0,C 180,E1 -13661.871,E2 -13661.871} C_VEL
LIN {X 0,Y 347.874,Z 397.154,A -85,B 0,C 180,E1 -13665.97,E2 -13665.97} C_VEL
LIN {X 0,Y 347.911,Z 397.151,A -85,B 0,C 180,E1 -13669.525,E2 -13669.525} C_VEL
LIN {X 0,Y 348.051,Z 397.13,A -85,B 0,C 180,E1 -13671.875,E2 -13671.875} C_VEL
LIN {X 0,Y 348.05,Z 397.131,A -85,B 0,C 180,E1 -13674.206,E2 -13674.206} C_VEL
LIN {X 0,Y 348.194,Z 397.115,A -85,B 0,C 180,E1 -13677.687,E2 -13677.687} C_VEL
LIN {X 0,Y 348.347,Z 397.095,A -85,B 0,C 180,E1 -13680,E2 -13680} C_VEL
LIN {X 0,Y 348.194,Z 397.114,A -85,B 0,C 180,E1 -13682.314,E2 -13682.314} C_VEL
LIN {X 0,Y 348.087,Z 397.121,A -85,B 0,C 180,E1 -13686.958,E2 -13686.958} C_VEL
LIN {X 0,Y 347.947,Z 397.139,A -85,B 0,C 180,E1 -13689.299,E2 -13689.299} C_VEL
LIN {X 0,Y 347.873,Z 397.149,A -85,B 0,C 180,E1 -13692.84,E2 -13692.84} C_VEL
LIN {X 0,Y 347.82,Z 397.158,A -85,B 0,C 180,E1 -13696.433,E2 -13696.433} C_VEL
LIN {X 0,Y 347.841,Z 397.152,A -85,B 0,C 180,E1 -13698.861,E2 -13698.861} C_VEL
LIN {X 0,Y 347.796,Z 397.158,A -85,B 0,C 180,E1 -13701.648,E2 -13701.648} C_VEL
LIN {X 0,Y 347.798,Z 397.161,A -85,B 0,C 180,E1 -13705.11,E2 -13705.11} C_VEL
LIN {X 0,Y 347.793,Z 397.16,A -85,B 0,C 180,E1 -13707.696,E2 -13707.696} C_VEL
LIN {X 0,Y 347.746,Z 397.166,A -85,B 0,C 180,E1 -13710.349,E2 -13710.349} C_VEL
LIN {X 0,Y 347.727,Z 397.171,A -85,B 0,C 180,E1 -13714.466,E2 -13714.466} C_VEL
LIN {X 0,Y 347.76,Z 397.168,A -85,B 0,C 180,E1 -13717.992,E2 -13717.992} C_VEL
LIN {X 0,Y 347.77,Z 397.168,A -85,B 0,C 180,E1 -13721.612,E2 -13721.612} C_VEL
LIN {X 0,Y 347.818,Z 397.158,A -85,B 0,C 180,E1 -13725.009,E2 -13725.009} C_VEL
LIN {X 0,Y 347.815,Z 397.227,A -85,B 0,C 180,E1 -13727.099,E2 -13727.099} C_VEL
LIN {X 0,Y 348.994,Z 403.127,A -85,B 0,C 180,E1 -13730.695,E2 -13730.695} C_VEL
LIN {X 0,Y 350.309,Z 409.943,A -85,B 0,C 180,E1 -13734.426,E2 -13734.426} C_VEL
LIN {X 0,Y 351.347,Z 415.564,A -85,B 0,C 180,E1 -13737.315,E2 -13737.315} C_VEL
LIN {X 0,Y 351.508,Z 418.481,A -85,B 0,C 180,E1 -13738.682,E2 -13738.682} C_VEL
LIN {X 0,Y 350.232,Z 426.05,A -85,B 0,C 180,E1 -13741.999,E2 -13741.999} C_VEL
LIN {X 0,Y 349.075,Z 434.727,A -85,B 0,C 180,E1 -13745.627,E2 -13745.627} C_VEL
LIN {X 0,Y 348.038,Z 444.214,A -85,B 0,C 180,E1 -13749.483,E2 -13749.483} C_VEL
LIN {X 0,Y 350.421,Z 457.175,A -85,B 0,C 180,E1 -13750.091,E2 -13750.091} C_VEL
LIN {X 0,Y 351.985,Z 469.79,A -85,B 0,C 180,E1 -13750.879,E2 -13750.879} C_VEL
LIN {X 0,Y 352.525,Z 480.459,A -85,B 0,C 180,E1 -13751.703,E2 -13751.703} C_VEL
LIN {X 0,Y 351.484,Z 491.509,A -85,B 0,C 180,E1 -13752.7,E2 -13752.7} C_VEL
LIN {X 0,Y 350.316,Z 501.712,A -85,B 0,C 180,E1 -13753.856,E2 -13753.856} C_VEL
LIN {X 0,Y 349.356,Z 510.645,A -85,B 0,C 180,E1 -13755.114,E2 -13755.114} C_VEL
LIN {X 0,Y 348.495,Z 519.201,A -85,B 0,C 180,E1 -13756.593,E2 -13756.593} C_VEL
LIN {X 0,Y 347.499,Z 527.382,A -85,B 0,C 180,E1 -13758.335,E2 -13758.335} C_VEL
LIN {X 0,Y 346.747,Z 536.38,A -85,B 0,C 180,E1 -13760.671,E2 -13760.671} C_VEL
LIN {X 0,Y 346.385,Z 541.758,A -85,B 0,C 180,E1 -13762.424,E2 -13762.424} C_VEL
LIN {X 0,Y 346.2,Z 545.915,A -85,B 0,C 180,E1 -13764.177,E2 -13764.177} C_VEL
LIN {X 0,Y 346.198,Z 548.072,A -85,B 0,C 180,E1 -13765.345,E2 -13765.345} C_VEL
LIN {X 0,Y 346.166,Z 549.746,A -85,B 0,C 180,E1 -13766.511,E2 -13766.511} C_VEL
LIN {X 0,Y 346.141,Z 551.001,A -85,B 0,C 180,E1 -13767.675,E2 -13767.675} C_VEL
LIN {X 0,Y 346.189,Z 551.835,A -85,B 0,C 180,E1 -13768.839,E2 -13768.839} C_VEL
LIN {X 0,Y 346.2,Z 552.211,A -85,B 0,C 180,E1 -13770.003,E2 -13770.003} C_VEL
LIN {X 0,Y 346.176,Z 552.184,A -85,B 0,C 180,E1 -13771.166,E2 -13771.166} C_VEL
LIN {X 0,Y 346.142,Z 551.758,A -85,B 0,C 180,E1 -13772.33,E2 -13772.33} C_VEL
LIN {X 0,Y 346.167,Z 550.898,A -85,B 0,C 180,E1 -13773.494,E2 -13773.494} C_VEL
LIN {X 0,Y 346.188,Z 549.604,A -85,B 0,C 180,E1 -13774.66,E2 -13774.66} C_VEL
LIN {X 0,Y 346.263,Z 546.873,A -85,B 0,C 180,E1 -13776.411,E2 -13776.411} C_VEL
LIN {X 0,Y 346.565,Z 543.106,A -85,B 0,C 180,E1 -13778.163,E2 -13778.163} C_VEL
LIN {X 0,Y 347.033,Z 538.202,A -85,B 0,C 180,E1 -13779.915,E2 -13779.915} C_VEL
LIN {X 0,Y 347.68,Z 532.025,A -85,B 0,C 180,E1 -13781.664,E2 -13781.664} C_VEL
LIN {X 0,Y 348.786,Z 524.386,A -85,B 0,C 180,E1 -13783.401,E2 -13783.401} C_VEL
LIN {X 0,Y 349.943,Z 514.865,A -85,B 0,C 180,E1 -13785.137,E2 -13785.137} C_VEL
LIN {X 0,Y 351.17,Z 505.113,A -85,B 0,C 180,E1 -13786.572,E2 -13786.572} C_VEL
LIN {X 0,Y 352.601,Z 494.234,A -85,B 0,C 180,E1 -13787.848,E2 -13787.848} C_VEL
LIN {X 0,Y 353.993,Z 482.104,A -85,B 0,C 180,E1 -13788.974,E2 -13788.974} C_VEL
LIN {X 0,Y 353.577,Z 470.211,A -85,B 0,C 180,E1 -13789.934,E2 -13789.934} C_VEL
LIN {X 0,Y 351.803,Z 456.762,A -85,B 0,C 180,E1 -13790.859,E2 -13790.859} C_VEL
LIN {X 0,Y 349.059,Z 443.533,A -85,B 0,C 180,E1 -13791.612,E2 -13791.612} C_VEL
LIN {X 0,Y 348.26,Z 439.586,A -85,B 0,C 180,E1 -13791.829,E2 -13791.829} C_VEL
LIN {X 0,Y 349.451,Z 428.565,A -85,B 0,C 180,E1 -13796.263,E2 -13796.263} C_VEL
LIN {X 0,Y 350.769,Z 419.337,A -85,B 0,C 180,E1 -13800.062,E2 -13800.062} C_VEL
LIN {X 0,Y 351.145,Z 416.251,A -85,B 0,C 180,E1 -13801.36,E2 -13801.36} C_VEL
LIN {X 0,Y 350.571,Z 411.584,A -85,B 0,C 180,E1 -13803.458,E2 -13803.458} C_VEL
LIN {X 0,Y 349.355,Z 405.353,A -85,B 0,C 180,E1 -13806.42,E2 -13806.42} C_VEL
LIN {X 0,Y 348.023,Z 398.423,A -85,B 0,C 180,E1 -13809.881,E2 -13809.881} C_VEL
LIN {X 0,Y 347.731,Z 397.171,A -85,B 0,C 180,E1 -13810.585,E2 -13810.585} C_VEL
LIN {X 0,Y 347.728,Z 397.172,A -85,B 0,C 180,E1 -13813.41,E2 -13813.41} C_VEL
LIN {X 0,Y 347.73,Z 397.164,A -85,B 0,C 180,E1 -13816.688,E2 -13816.688} C_VEL
LIN {X 0,Y 347.708,Z 397.171,A -85,B 0,C 180,E1 -13820.183,E2 -13820.183} C_VEL
LIN {X 0,Y 347.764,Z 397.162,A -85,B 0,C 180,E1 -13822.679,E2 -13822.679} C_VEL
LIN {X 0,Y 347.757,Z 397.167,A -85,B 0,C 180,E1 -13825.957,E2 -13825.957} C_VEL
LIN {X 0,Y 347.746,Z 397.171,A -85,B 0,C 180,E1 -13829.651,E2 -13829.651} C_VEL
LIN {X 0,Y 347.741,Z 397.17,A -85,B 0,C 180,E1 -13833.6,E2 -13833.6} C_VEL
LIN {X 0,Y 347.756,Z 397.166,A -85,B 0,C 180,E1 -13836.159,E2 -13836.159} C_VEL
LIN {X 0,Y 347.813,Z 397.161,A -85,B 0,C 180,E1 -13839.909,E2 -13839.909} C_VEL
LIN {X 0,Y 347.874,Z 397.155,A -85,B 0,C 180,E1 -13842.359,E2 -13842.359} C_VEL
LIN {X 0,Y 347.906,Z 397.149,A -85,B 0,C 180,E1 -13845.971,E2 -13845.971} C_VEL
LIN {X 0,Y 347.9,Z 397.15,A -85,B 0,C 180,E1 -13849.524,E2 -13849.524} C_VEL
LIN {X 0,Y 348.051,Z 397.331,A -85,B 0,C 180,E1 -13851.874,E2 -13851.874} C_VEL
LIN {X 0,Y 348.784,Z 401.291,A -85,B 0,C 180,E1 -13854.217,E2 -13854.217} C_VEL
LIN {X 0,Y 349.05,Z 405.317,A -85,B 0,C 180,E1 -13856.537,E2 -13856.537} C_VEL
LIN {X 0,Y 348.843,Z 410.574,A -85,B 0,C 180,E1 -13859.422,E2 -13859.422} C_VEL
LIN {X 0,Y 348.214,Z 419.153,A -85,B 0,C 180,E1 -13864.05,E2 -13864.05} C_VEL
LIN {X 0,Y 347.994,Z 424.475,A -85,B 0,C 180,E1 -13866.959,E2 -13866.959} C_VEL
LIN {X 0,Y 347.765,Z 428.391,A -85,B 0,C 180,E1 -13869.084,E2 -13869.084} C_VEL
LIN {X 0,Y 352.271,Z 443.788,A -85,B 0,C 180,E1 -13870.184,E2 -13870.184} C_VEL
LIN {X 0,Y 354.63,Z 455.612,A -85,B 0,C 180,E1 -13871.141,E2 -13871.141} C_VEL
LIN {X 0,Y 355.343,Z 461.136,A -85,B 0,C 180,E1 -13871.634,E2 -13871.634} C_VEL
LIN {X 0,Y 354.026,Z 473.749,A -85,B 0,C 180,E1 -13872.747,E2 -13872.747} C_VEL
LIN {X 0,Y 352.709,Z 484.667,A -85,B 0,C 180,E1 -13873.981,E2 -13873.981} C_VEL
LIN {X 0,Y 351.233,Z 495.8,A -85,B 0,C 180,E1 -13875.558,E2 -13875.558} C_VEL
LIN {X 0,Y 350.118,Z 503.62,A -85,B 0,C 180,E1 -13876.921,E2 -13876.921} C_VEL
LIN {X 0,Y 348.888,Z 512.303,A -85,B 0,C 180,E1 -13878.802,E2 -13878.802} C_VEL
LIN {X 0,Y 347.914,Z 519.253,A -85,B 0,C 180,E1 -13880.702,E2 -13880.702} C_VEL
LIN {X 0,Y 347.104,Z 524.672,A -85,B 0,C 180,E1 -13882.625,E2 -13882.625} C_VEL
LIN {X 0,Y 346.727,Z 528.088,A -85,B 0,C 180,E1 -13884.196,E2 -13884.196} C_VEL
LIN {X 0,Y 346.538,Z 529.822,A -85,B 0,C 180,E1 -13885.207,E2 -13885.207} C_VEL
LIN {X 0,Y 346.225,Z 531.85,A -85,B 0,C 180,E1 -13886.725,E2 -13886.725} C_VEL
LIN {X 0,Y 346.066,Z 532.875,A -85,B 0,C 180,E1 -13887.845,E2 -13887.845} C_VEL
LIN {X 0,Y 345.941,Z 533.597,A -85,B 0,C 180,E1 -13889.181,E2 -13889.181} C_VEL
LIN {X 0,Y 345.901,Z 533.644,A -85,B 0,C 180,E1 -13891.419,E2 -13891.419} C_VEL
LIN {X 0,Y 345.932,Z 532.205,A -85,B 0,C 180,E1 -13893.593,E2 -13893.593} C_VEL
LIN {X 0,Y 346.203,Z 529.438,A -85,B 0,C 180,E1 -13895.705,E2 -13895.705} C_VEL
LIN {X 0,Y 346.547,Z 525.398,A -85,B 0,C 180,E1 -13897.726,E2 -13897.726} C_VEL
LIN {X 0,Y 346.951,Z 520.097,A -85,B 0,C 180,E1 -13899.667,E2 -13899.667} C_VEL
LIN {X 0,Y 347.591,Z 513.388,A -85,B 0,C 180,E1 -13901.571,E2 -13901.571} C_VEL
LIN {X 0,Y 348.398,Z 505.027,A -85,B 0,C 180,E1 -13903.429,E2 -13903.429} C_VEL
LIN {X 0,Y 349.328,Z 496.112,A -85,B 0,C 180,E1 -13905.02,E2 -13905.02} C_VEL
LIN {X 0,Y 350.279,Z 486.109,A -85,B 0,C 180,E1 -13906.467,E2 -13906.467} C_VEL
LIN {X 0,Y 351.32,Z 475.104,A -85,B 0,C 180,E1 -13907.745,E2 -13907.745} C_VEL
LIN {X 0,Y 352.262,Z 463.472,A -85,B 0,C 180,E1 -13908.821,E2 -13908.821} C_VEL
LIN {X 0,Y 352.567,Z 457.1,A -85,B 0,C 180,E1 -13909.307,E2 -13909.307} C_VEL
LIN {X 0,Y 350.494,Z 444.471,A -85,B 0,C 180,E1 -13910.207,E2 -13910.207} C_VEL
LIN {X 0,Y 347.884,Z 431.646,A -85,B 0,C 180,E1 -13910.913,E2 -13910.913} C_VEL
LIN {X 0,Y 347.039,Z 427.335,A -85,B 0,C 180,E1 -13911.11,E2 -13911.11} C_VEL
LIN {X 0,Y 347.329,Z 420.505,A -85,B 0,C 180,E1 -13914.78,E2 -13914.78} C_VEL
LIN {X 0,Y 347.543,Z 414.026,A -85,B 0,C 180,E1 -13918.278,E2 -13918.278} C_VEL
LIN {X 0,Y 347.83,Z 407.791,A -85,B 0,C 180,E1 -13921.65,E2 -13921.65} C_VEL
LIN {X 0,Y 348.103,Z 401.066,A -85,B 0,C 180,E1 -13925.301,E2 -13925.301} C_VEL
LIN {X 0,Y 347.894,Z 397.153,A -85,B 0,C 180,E1 -13927.46,E2 -13927.46} C_VEL
LIN {X 0,Y 347.893,Z 397.152,A -85,B 0,C 180,E1 -13931.708,E2 -13931.708} C_VEL
LIN {X 0,Y 347.899,Z 397.149,A -85,B 0,C 180,E1 -13935.969,E2 -13935.969} C_VEL
LIN {X 0,Y 347.929,Z 397.148,A -85,B 0,C 180,E1 -13939.523,E2 -13939.523} C_VEL
LIN {X 0,Y 348.068,Z 397.131,A -85,B 0,C 180,E1 -13943.039,E2 -13943.039} C_VEL
LIN {X 0,Y 348.095,Z 397.131,A -85,B 0,C 180,E1 -13947.394,E2 -13947.394} C_VEL
LIN {X 0,Y 348.552,Z 400.662,A -85,B 0,C 180,E1 -13949.997,E2 -13949.997} C_VEL
LIN {X 0,Y 347.956,Z 405.689,A -85,B 0,C 180,E1 -13953.471,E2 -13953.471} C_VEL
LIN {X 0,Y 347.911,Z 409.063,A -85,B 0,C 180,E1 -13955.794,E2 -13955.794} C_VEL
LIN {X 0,Y 347.475,Z 414.32,A -85,B 0,C 180,E1 -13959.309,E2 -13959.309} C_VEL
LIN {X 0,Y 347.171,Z 419.726,A -85,B 0,C 180,E1 -13962.864,E2 -13962.864} C_VEL
LIN {X 0,Y 346.866,Z 424.971,A -85,B 0,C 180,E1 -13966.249,E2 -13966.249} C_VEL
LIN {X 0,Y 349.363,Z 437.478,A -85,B 0,C 180,E1 -13966.956,E2 -13966.956} C_VEL
LIN {X 0,Y 351.161,Z 448.203,A -85,B 0,C 180,E1 -13967.768,E2 -13967.768} C_VEL
LIN {X 0,Y 351.528,Z 451.434,A -85,B 0,C 180,E1 -13968.049,E2 -13968.049} C_VEL
LIN {X 0,Y 350.675,Z 462.119,A -85,B 0,C 180,E1 -13969.052,E2 -13969.052} C_VEL
LIN {X 0,Y 349.809,Z 472.13,A -85,B 0,C 180,E1 -13970.274,E2 -13970.274} C_VEL
LIN {X 0,Y 349.114,Z 480.062,A -85,B 0,C 180,E1 -13971.487,E2 -13971.487} C_VEL
LIN {X 0,Y 348.368,Z 487.272,A -85,B 0,C 180,E1 -13972.849,E2 -13972.849} C_VEL
LIN {X 0,Y 347.675,Z 494.419,A -85,B 0,C 180,E1 -13974.545,E2 -13974.545} C_VEL
LIN {X 0,Y 347.049,Z 500.493,A -85,B 0,C 180,E1 -13976.453,E2 -13976.453} C_VEL
LIN {X 0,Y 346.651,Z 505.009,A -85,B 0,C 180,E1 -13978.449,E2 -13978.449} C_VEL
LIN {X 0,Y 346.341,Z 507.967,A -85,B 0,C 180,E1 -13980.481,E2 -13980.481} C_VEL
LIN {X 0,Y 346.217,Z 509.107,A -85,B 0,C 180,E1 -13981.852,E2 -13981.852} C_VEL
LIN {X 0,Y 346.211,Z 509.536,A -85,B 0,C 180,E1 -13983.666,E2 -13983.666} C_VEL
LIN {X 0,Y 346.408,Z 508.604,A -85,B 0,C 180,E1 -13985.755,E2 -13985.755} C_VEL
LIN {X 0,Y 346.76,Z 506.168,A -85,B 0,C 180,E1 -13987.774,E2 -13987.774} C_VEL
LIN {X 0,Y 347.284,Z 502.27,A -85,B 0,C 180,E1 -13989.736,E2 -13989.736} C_VEL
LIN {X 0,Y 347.342,Z 501.818,A -85,B 0,C 180,E1 -13989.915,E2 -13989.915} C_VEL
LIN {X 0,Y 346.991,Z 499.545,A -85,B 0,C 180,E1 -13990.812,E2 -13990.812} C_VEL
LIN {X 0,Y 344.702,Z 495.392,A -85,B 0,C 180,E1 -13992.261,E2 -13992.261} C_VEL
LIN {X 0,Y 342.507,Z 490.536,A -85,B 0,C 180,E1 -13993.657,E2 -13993.657} C_VEL
LIN {X 0,Y 342.297,Z 487.066,A -85,B 0,C 180,E1 -13994.456,E2 -13994.456} C_VEL
LIN {X 0,Y 343.256,Z 479.463,A -85,B 0,C 180,E1 -13995.883,E2 -13995.883} C_VEL
LIN {X 0,Y 344.432,Z 470.166,A -85,B 0,C 180,E1 -13997.265,E2 -13997.265} C_VEL
LIN {X 0,Y 345.515,Z 459.741,A -85,B 0,C 180,E1 -13998.475,E2 -13998.475} C_VEL
LIN {X 0,Y 345.9,Z 453.273,A -85,B 0,C 180,E1 -13999.092,E2 -13999.092} C_VEL
LIN {X 0,Y 344.341,Z 443.271,A -85,B 0,C 180,E1 -14000.001,E2 -14000.001} C_VEL
LIN {X 0,Y 341.664,Z 431.894,A -85,B 0,C 180,E1 -14000.859,E2 -14000.859} C_VEL
LIN {X 0,Y 340.187,Z 426.103,A -85,B 0,C 180,E1 -14001.228,E2 -14001.228} C_VEL
LIN {X 0,Y 340.482,Z 421.093,A -85,B 0,C 180,E1 -14004.694,E2 -14004.694} C_VEL
LIN {X 0,Y 340.746,Z 416.776,A -85,B 0,C 180,E1 -14007.733,E2 -14007.733} C_VEL
LIN {X 0,Y 341.195,Z 411.29,A -85,B 0,C 180,E1 -14011.722,E2 -14011.722} C_VEL
LIN {X 0,Y 341.588,Z 407.134,A -85,B 0,C 180,E1 -14014.851,E2 -14014.851} C_VEL
LIN {X 0,Y 341.497,Z 402.74,A -85,B 0,C 180,E1 -14018.258,E2 -14018.258} C_VEL
LIN {X 0,Y 340.873,Z 398.387,A -85,B 0,C 180,E1 -14021.985,E2 -14021.985} C_VEL
LIN {X 0,Y 340.785,Z 398.042,A -85,B 0,C 180,E1 -14022.601,E2 -14022.601} C_VEL
LIN {X 0,Y 340.846,Z 398.03,A -85,B 0,C 180,E1 -14025.704,E2 -14025.704} C_VEL
LIN {X 0,Y 340.854,Z 398.029,A -85,B 0,C 180,E1 -14029.306,E2 -14029.306} C_VEL
LIN {X 0,Y 341.055,Z 398.006,A -85,B 0,C 180,E1 -14032.898,E2 -14032.898} C_VEL
LIN {X 0,Y 341.157,Z 397.992,A -85,B 0,C 180,E1 -14037.639,E2 -14037.639} C_VEL
LIN {X 0,Y 341.317,Z 397.97,A -85,B 0,C 180,E1 -14040,E2 -14040} C_VEL
LIN {X 0,Y 341.157,Z 397.991,A -85,B 0,C 180,E1 -14042.362,E2 -14042.362} C_VEL
LIN {X 0,Y 341.056,Z 397.998,A -85,B 0,C 180,E1 -14047.103,E2 -14047.103} C_VEL
LIN {X 0,Y 340.854,Z 398.027,A -85,B 0,C 180,E1 -14050.695,E2 -14050.695} C_VEL
LIN {X 0,Y 340.841,Z 398.029,A -85,B 0,C 180,E1 -14054.326,E2 -14054.326} C_VEL
LIN {X 0,Y 340.818,Z 398.026,A -85,B 0,C 180,E1 -14058.469,E2 -14058.469} C_VEL
LIN {X 0,Y 340.736,Z 398.038,A -85,B 0,C 180,E1 -14061.86,E2 -14061.86} C_VEL
LIN {X 0,Y 340.756,Z 398.04,A -85,B 0,C 180,E1 -14065.666,E2 -14065.666} C_VEL
LIN {X 0,Y 340.723,Z 398.043,A -85,B 0,C 180,E1 -14068.322,E2 -14068.322} C_VEL
LIN {X 0,Y 340.686,Z 398.048,A -85,B 0,C 180,E1 -14071.046,E2 -14071.046} C_VEL
LIN {X 0,Y 340.701,Z 398.047,A -85,B 0,C 180,E1 -14075.281,E2 -14075.281} C_VEL
LIN {X 0,Y 340.702,Z 398.047,A -85,B 0,C 180,E1 -14078.39,E2 -14078.39} C_VEL
LIN {X 0,Y 340.711,Z 398.047,A -85,B 0,C 180,E1 -14081.306,E2 -14081.306} C_VEL
LIN {X 0,Y 340.768,Z 398.04,A -85,B 0,C 180,E1 -14084.525,E2 -14084.525} C_VEL
LIN {X 0,Y 340.778,Z 398.203,A -85,B 0,C 180,E1 -14086.449,E2 -14086.449} C_VEL
LIN {X 0,Y 341.753,Z 403.029,A -85,B 0,C 180,E1 -14089.543,E2 -14089.543} C_VEL
LIN {X 0,Y 342.92,Z 409.09,A -85,B 0,C 180,E1 -14093.063,E2 -14093.063} C_VEL
LIN {X 0,Y 344.295,Z 416.161,A -85,B 0,C 180,E1 -14096.817,E2 -14096.817} C_VEL
LIN {X 0,Y 344.563,Z 419.673,A -85,B 0,C 180,E1 -14098.565,E2 -14098.565} C_VEL
LIN {X 0,Y 343.028,Z 428.648,A -85,B 0,C 180,E1 -14102.553,E2 -14102.553} C_VEL
LIN {X 0,Y 341.811,Z 437.581,A -85,B 0,C 180,E1 -14106.366,E2 -14106.366} C_VEL
LIN {X 0,Y 341.075,Z 444.073,A -85,B 0,C 180,E1 -14109.025,E2 -14109.025} C_VEL
LIN {X 0,Y 343.613,Z 457.465,A -85,B 0,C 180,E1 -14109.685,E2 -14109.685} C_VEL
LIN {X 0,Y 345.167,Z 470.104,A -85,B 0,C 180,E1 -14110.509,E2 -14110.509} C_VEL
LIN {X 0,Y 345.709,Z 480.378,A -85,B 0,C 180,E1 -14111.329,E2 -14111.329} C_VEL
LIN {X 0,Y 344.862,Z 489.952,A -85,B 0,C 180,E1 -14112.204,E2 -14112.204} C_VEL
LIN {X 0,Y 343.488,Z 501.425,A -85,B 0,C 180,E1 -14113.511,E2 -14113.511} C_VEL
LIN {X 0,Y 342.392,Z 511.118,A -85,B 0,C 180,E1 -14114.921,E2 -14114.921} C_VEL
LIN {X 0,Y 341.39,Z 520.44,A -85,B 0,C 180,E1 -14116.612,E2 -14116.612} C_VEL
LIN {X 0,Y 340.389,Z 528.28,A -85,B 0,C 180,E1 -14118.39,E2 -14118.39} C_VEL
LIN {X 0,Y 339.574,Z 537.871,A -85,B 0,C 180,E1 -14121.073,E2 -14121.073} C_VEL
LIN {X 0,Y 339.248,Z 542.87,A -85,B 0,C 180,E1 -14122.863,E2 -14122.863} C_VEL
LIN {X 0,Y 339.11,Z 545.754,A -85,B 0,C 180,E1 -14124.154,E2 -14124.154} C_VEL
LIN {X 0,Y 339.093,Z 547.75,A -85,B 0,C 180,E1 -14125.247,E2 -14125.247} C_VEL
LIN {X 0,Y 339.09,Z 549.449,A -85,B 0,C 180,E1 -14126.438,E2 -14126.438} C_VEL
LIN {X 0,Y 339.051,Z 550.727,A -85,B 0,C 180,E1 -14127.627,E2 -14127.627} C_VEL
LIN {X 0,Y 339.09,Z 551.595,A -85,B 0,C 180,E1 -14128.815,E2 -14128.815} C_VEL
LIN {X 0,Y 339.103,Z 552.004,A -85,B 0,C 180,E1 -14130.003,E2 -14130.003} C_VEL
LIN {X 0,Y 339.076,Z 552,A -85,B 0,C 180,E1 -14131.19,E2 -14131.19} C_VEL
LIN {X 0,Y 339.053,Z 551.595,A -85,B 0,C 180,E1 -14132.379,E2 -14132.379} C_VEL
LIN {X 0,Y 339.09,Z 550.777,A -85,B 0,C 180,E1 -14133.567,E2 -14133.567} C_VEL
LIN {X 0,Y 339.116,Z 547.968,A -85,B 0,C 180,E1 -14135.856,E2 -14135.856} C_VEL
LIN {X 0,Y 339.401,Z 544.451,A -85,B 0,C 180,E1 -14137.738,E2 -14137.738} C_VEL
LIN {X 0,Y 339.852,Z 540,A -85,B 0,C 180,E1 -14139.525,E2 -14139.525} C_VEL
LIN {X 0,Y 340.515,Z 534.355,A -85,B 0,C 180,E1 -14141.31,E2 -14141.31} C_VEL
LIN {X 0,Y 341.485,Z 527.319,A -85,B 0,C 180,E1 -14143.087,E2 -14143.087} C_VEL
LIN {X 0,Y 342.716,Z 518.568,A -85,B 0,C 180,E1 -14144.855,E2 -14144.855} C_VEL
LIN {X 0,Y 343.77,Z 510.174,A -85,B 0,C 180,E1 -14146.247,E2 -14146.247} C_VEL
LIN {X 0,Y 345.199,Z 499.935,A -85,B 0,C 180,E1 -14147.631,E2 -14147.631} C_VEL
LIN {X 0,Y 346.677,Z 489.288,A -85,B 0,C 180,E1 -14148.776,E2 -14148.776} C_VEL
LIN {X 0,Y 347.342,Z 481.397,A -85,B 0,C 180,E1 -14149.505,E2 -14149.505} C_VEL
LIN {X 0,Y 346.835,Z 469.414,A -85,B 0,C 180,E1 -14150.501,E2 -14150.501} C_VEL
LIN {X 0,Y 345.033,Z 456.26,A -85,B 0,C 180,E1 -14151.435,E2 -14151.435} C_VEL
LIN {X 0,Y 342.216,Z 442.855,A -85,B 0,C 180,E1 -14152.223,E2 -14152.223} C_VEL
LIN {X 0,Y 341.325,Z 438.782,A -85,B 0,C 180,E1 -14152.472,E2 -14152.472} C_VEL
LIN {X 0,Y 342.593,Z 428.22,A -85,B 0,C 180,E1 -14156.83,E2 -14156.83} C_VEL
LIN {X 0,Y 343.968,Z 419.001,A -85,B 0,C 180,E1 -14160.72,E2 -14160.72} C_VEL
LIN {X 0,Y 344.092,Z 415.94,A -85,B 0,C 180,E1 -14162.078,E2 -14162.078} C_VEL
LIN {X 0,Y 343.012,Z 409.727,A -85,B 0,C 180,E1 -14165.01,E2 -14165.01} C_VEL
LIN {X 0,Y 341.434,Z 401.664,A -85,B 0,C 180,E1 -14169.053,E2 -14169.053} C_VEL
LIN {X 0,Y 340.706,Z 398.046,A -85,B 0,C 180,E1 -14171.026,E2 -14171.026} C_VEL
LIN {X 0,Y 340.644,Z 398.053,A -85,B 0,C 180,E1 -14174.547,E2 -14174.547} C_VEL
LIN {X 0,Y 340.699,Z 398.046,A -85,B 0,C 180,E1 -14177.957,E2 -14177.957} C_VEL
LIN {X 0,Y 340.727,Z 398.035,A -85,B 0,C 180,E1 -14181.771,E2 -14181.771} C_VEL
LIN {X 0,Y 340.731,Z 398.042,A -85,B 0,C 180,E1 -14185.596,E2 -14185.596} C_VEL
LIN {X 0,Y 340.701,Z 398.044,A -85,B 0,C 180,E1 -14188.955,E2 -14188.955} C_VEL
LIN {X 0,Y 340.717,Z 398.045,A -85,B 0,C 180,E1 -14193.012,E2 -14193.012} C_VEL
LIN {X 0,Y 340.708,Z 398.047,A -85,B 0,C 180,E1 -14196.925,E2 -14196.925} C_VEL
LIN {X 0,Y 340.796,Z 398.036,A -85,B 0,C 180,E1 -14200.733,E2 -14200.733} C_VEL
LIN {X 0,Y 340.794,Z 398.037,A -85,B 0,C 180,E1 -14203.219,E2 -14203.219} C_VEL
LIN {X 0,Y 340.85,Z 398.031,A -85,B 0,C 180,E1 -14206.89,E2 -14206.89} C_VEL
LIN {X 0,Y 340.942,Z 398.163,A -85,B 0,C 180,E1 -14211.166,E2 -14211.166} C_VEL
LIN {X 0,Y 341.891,Z 402.893,A -85,B 0,C 180,E1 -14214.1,E2 -14214.1} C_VEL
LIN {X 0,Y 342.174,Z 406.92,A -85,B 0,C 180,E1 -14216.467,E2 -14216.467} C_VEL
LIN {X 0,Y 341.916,Z 412.236,A -85,B 0,C 180,E1 -14219.411,E2 -14219.411} C_VEL
LIN {X 0,Y 341.242,Z 420.759,A -85,B 0,C 180,E1 -14224.133,E2 -14224.133} C_VEL
LIN {X 0,Y 340.998,Z 426.112,A -85,B 0,C 180,E1 -14227.103,E2 -14227.103} C_VEL
LIN {X 0,Y 340.842,Z 428.698,A -85,B 0,C 180,E1 -14228.489,E2 -14228.489} C_VEL
LIN {X 0,Y 344.919,Z 442.016,A -85,B 0,C 180,E1 -14229.465,E2 -14229.465} C_VEL
LIN {X 0,Y 347.647,Z 454.124,A -85,B 0,C 180,E1 -14230.483,E2 -14230.483} C_VEL
LIN {X 0,Y 348.74,Z 462.11,A -85,B 0,C 180,E1 -14231.213,E2 -14231.213} C_VEL
LIN {X 0,Y 347.527,Z 473.659,A -85,B 0,C 180,E1 -14232.259,E2 -14232.259} C_VEL
LIN {X 0,Y 346.28,Z 483.57,A -85,B 0,C 180,E1 -14233.375,E2 -14233.375} C_VEL
LIN {X 0,Y 344.84,Z 493.543,A -85,B 0,C 180,E1 -14234.759,E2 -14234.759} C_VEL
LIN {X 0,Y 343.547,Z 502.423,A -85,B 0,C 180,E1 -14236.279,E2 -14236.279} C_VEL
LIN {X 0,Y 342.379,Z 510.303,A -85,B 0,C 180,E1 -14237.933,E2 -14237.933} C_VEL
LIN {X 0,Y 341.204,Z 517.693,A -85,B 0,C 180,E1 -14239.868,E2 -14239.868} C_VEL
LIN {X 0,Y 340.356,Z 523.503,A -85,B 0,C 180,E1 -14241.819,E2 -14241.819} C_VEL
LIN {X 0,Y 339.729,Z 527.92,A -85,B 0,C 180,E1 -14243.771,E2 -14243.771} C_VEL
LIN {X 0,Y 339.302,Z 531.151,A -85,B 0,C 180,E1 -14245.783,E2 -14245.783} C_VEL
LIN {X 0,Y 339.059,Z 532.605,A -85,B 0,C 180,E1 -14247.13,E2 -14247.13} C_VEL
LIN {X 0,Y 338.823,Z 533.92,A -85,B 0,C 180,E1 -14249.401,E2 -14249.401} C_VEL
LIN {X 0,Y 338.781,Z 533.677,A -85,B 0,C 180,E1 -14251.726,E2 -14251.726} C_VEL
LIN {X 0,Y 338.874,Z 531.921,A -85,B 0,C 180,E1 -14254.053,E2 -14254.053} C_VEL
LIN {X 0,Y 339.202,Z 529.004,A -85,B 0,C 180,E1 -14256.092,E2 -14256.092} C_VEL
LIN {X 0,Y 339.536,Z 524.749,A -85,B 0,C 180,E1 -14258.133,E2 -14258.133} C_VEL
LIN {X 0,Y 339.986,Z 519.246,A -85,B 0,C 180,E1 -14260.104,E2 -14260.104} C_VEL
LIN {X 0,Y 340.669,Z 512.242,A -85,B 0,C 180,E1 -14262.037,E2 -14262.037} C_VEL
LIN {X 0,Y 341.529,Z 503.614,A -85,B 0,C 180,E1 -14263.924,E2 -14263.924} C_VEL
LIN {X 0,Y 342.493,Z 494.93,A -85,B 0,C 180,E1 -14265.447,E2 -14265.447} C_VEL
LIN {X 0,Y 343.596,Z 484.045,A -85,B 0,C 180,E1 -14266.99,E2 -14266.99} C_VEL
LIN {X 0,Y 344.601,Z 473.438,A -85,B 0,C 180,E1 -14268.199,E2 -14268.199} C_VEL
LIN {X 0,Y 345.611,Z 460.664,A -85,B 0,C 180,E1 -14269.338,E2 -14269.338} C_VEL
LIN {X 0,Y 345.467,Z 456.965,A -85,B 0,C 180,E1 -14269.632,E2 -14269.632} C_VEL
LIN {X 0,Y 343.259,Z 443.578,A -85,B 0,C 180,E1 -14270.6,E2 -14270.6} C_VEL
LIN {X 0,Y 340.585,Z 430.424,A -85,B 0,C 180,E1 -14271.312,E2 -14271.312} C_VEL
LIN {X 0,Y 339.995,Z 427.419,A -85,B 0,C 180,E1 -14271.483,E2 -14271.483} C_VEL
LIN {X 0,Y 340.27,Z 421.567,A -85,B 0,C 180,E1 -14274.666,E2 -14274.666} C_VEL
LIN {X 0,Y 340.516,Z 414.764,A -85,B 0,C 180,E1 -14278.377,E2 -14278.377} C_VEL
LIN {X 0,Y 340.808,Z 408.716,A -85,B 0,C 180,E1 -14281.684,E2 -14281.684} C_VEL
LIN {X 0,Y 341.087,Z 401.492,A -85,B 0,C 180,E1 -14285.661,E2 -14285.661} C_VEL
LIN {X 0,Y 340.865,Z 398.028,A -85,B 0,C 180,E1 -14287.663,E2 -14287.663} C_VEL
LIN {X 0,Y 340.86,Z 398.028,A -85,B 0,C 180,E1 -14291.982,E2 -14291.982} C_VEL
LIN {X 0,Y 340.871,Z 398.025,A -85,B 0,C 180,E1 -14295.703,E2 -14295.703} C_VEL
LIN {X 0,Y 340.872,Z 398.026,A -85,B 0,C 180,E1 -14299.304,E2 -14299.304} C_VEL
LIN {X 0,Y 341.016,Z 398.008,A -85,B 0,C 180,E1 -14302.894,E2 -14302.894} C_VEL
LIN {X 0,Y 340.819,Z 398.036,A -85,B 0,C 180,E1 -14305.266,E2 -14305.266} C_VEL
LIN {X 0,Y 341.006,Z 398.037,A -85,B 0,C 180,E1 -14307.192,E2 -14307.192} C_VEL
LIN {X 0,Y 341.452,Z 400.17,A -85,B 0,C 180,E1 -14308.818,E2 -14308.818} C_VEL
LIN {X 0,Y 341.355,Z 403.433,A -85,B 0,C 180,E1 -14311.177,E2 -14311.177} C_VEL
LIN {X 0,Y 340.876,Z 410.227,A -85,B 0,C 180,E1 -14315.914,E2 -14315.914} C_VEL
LIN {X 0,Y 340.405,Z 415.486,A -85,B 0,C 180,E1 -14319.504,E2 -14319.504} C_VEL
LIN {X 0,Y 340.064,Z 420.964,A -85,B 0,C 180,E1 -14323.137,E2 -14323.137} C_VEL
LIN {X 0,Y 339.807,Z 425.189,A -85,B 0,C 180,E1 -14325.902,E2 -14325.902} C_VEL
LIN {X 0,Y 342.139,Z 436.621,A -85,B 0,C 180,E1 -14326.556,E2 -14326.556} C_VEL
LIN {X 0,Y 344.053,Z 447.475,A -85,B 0,C 180,E1 -14327.379,E2 -14327.379} C_VEL
LIN {X 0,Y 344.619,Z 452.343,A -85,B 0,C 180,E1 -14327.809,E2 -14327.809} C_VEL
LIN {X 0,Y 343.777,Z 462.415,A -85,B 0,C 180,E1 -14328.78,E2 -14328.78} C_VEL
LIN {X 0,Y 342.924,Z 471.789,A -85,B 0,C 180,E1 -14329.937,E2 -14329.937} C_VEL
LIN {X 0,Y 342.095,Z 481.044,A -85,B 0,C 180,E1 -14331.383,E2 -14331.383} C_VEL
LIN {X 0,Y 341.167,Z 489.38,A -85,B 0,C 180,E1 -14333.038,E2 -14333.038} C_VEL
LIN {X 0,Y 340.495,Z 496.018,A -85,B 0,C 180,E1 -14334.746,E2 -14334.746} C_VEL
LIN {X 0,Y 340.005,Z 500.983,A -85,B 0,C 180,E1 -14336.382,E2 -14336.382} C_VEL
LIN {X 0,Y 339.68,Z 504.214,A -85,B 0,C 180,E1 -14337.764,E2 -14337.764} C_VEL
LIN {X 0,Y 339.361,Z 507.594,A -85,B 0,C 180,E1 -14339.8,E2 -14339.8} C_VEL
LIN {X 0,Y 339.153,Z 509.496,A -85,B 0,C 180,E1 -14341.831,E2 -14341.831} C_VEL
LIN {X 0,Y 339.156,Z 509.917,A -85,B 0,C 180,E1 -14344.017,E2 -14344.017} C_VEL
LIN {X 0,Y 339.392,Z 508.755,A -85,B 0,C 180,E1 -14346.139,E2 -14346.139} C_VEL
LIN {X 0,Y 339.825,Z 505.883,A -85,B 0,C 180,E1 -14348.344,E2 -14348.344} C_VEL
LIN {X 0,Y 340.375,Z 502.063,A -85,B 0,C 180,E1 -14350.185,E2 -14350.185} C_VEL
LIN {X 0,Y 341.068,Z 496.486,A -85,B 0,C 180,E1 -14352.115,E2 -14352.115} C_VEL
LIN {X 0,Y 341.875,Z 490.473,A -85,B 0,C 180,E1 -14353.705,E2 -14353.705} C_VEL
LIN {X 0,Y 342.297,Z 487.066,A -85,B 0,C 180,E1 -14354.456,E2 -14354.456} C_VEL
LIN {X 0,Y 342.135,Z 483.369,A -85,B 0,C 180,E1 -14355.228,E2 -14355.228} C_VEL
LIN {X 0,Y 340.198,Z 477.063,A -85,B 0,C 180,E1 -14356.478,E2 -14356.478} C_VEL
LIN {X 0,Y 338.314,Z 470.179,A -85,B 0,C 180,E1 -14357.637,E2 -14357.637} C_VEL
LIN {X 0,Y 338.217,Z 465.547,A -85,B 0,C 180,E1 -14358.255,E2 -14358.255} C_VEL
LIN {X 0,Y 339.24,Z 456.001,A -85,B 0,C 180,E1 -14359.264,E2 -14359.264} C_VEL
LIN {X 0,Y 337.956,Z 446.304,A -85,B 0,C 180,E1 -14360.21,E2 -14360.21} C_VEL
LIN {X 0,Y 335.454,Z 434.886,A -85,B 0,C 180,E1 -14361.141,E2 -14361.141} C_VEL
LIN {X 0,Y 333.225,Z 426.312,A -85,B 0,C 180,E1 -14361.741,E2 -14361.741} C_VEL
LIN {X 0,Y 333.493,Z 421.266,A -85,B 0,C 180,E1 -14365.32,E2 -14365.32} C_VEL
LIN {X 0,Y 333.765,Z 417.225,A -85,B 0,C 180,E1 -14368.237,E2 -14368.237} C_VEL
LIN {X 0,Y 334.325,Z 411.56,A -85,B 0,C 180,E1 -14372.454,E2 -14372.454} C_VEL
LIN {X 0,Y 334.596,Z 408.003,A -85,B 0,C 180,E1 -14375.16,E2 -14375.16} C_VEL
LIN {X 0,Y 334.576,Z 404.719,A -85,B 0,C 180,E1 -14377.784,E2 -14377.784} C_VEL
LIN {X 0,Y 334.093,Z 400.777,A -85,B 0,C 180,E1 -14381.183,E2 -14381.183} C_VEL
LIN {X 0,Y 333.733,Z 398.922,A -85,B 0,C 180,E1 -14383.011,E2 -14383.011} C_VEL
LIN {X 0,Y 333.776,Z 398.911,A -85,B 0,C 180,E1 -14386.608,E2 -14386.608} C_VEL
LIN {X 0,Y 333.842,Z 398.901,A -85,B 0,C 180,E1 -14390.305,E2 -14390.305} C_VEL
LIN {X 0,Y 334.004,Z 398.883,A -85,B 0,C 180,E1 -14392.747,E2 -14392.747} C_VEL
LIN {X 0,Y 334.118,Z 398.868,A -85,B 0,C 180,E1 -14397.589,E2 -14397.589} C_VEL
LIN {X 0,Y 334.266,Z 398.849,A -85,B 0,C 180,E1 -14400,E2 -14400} C_VEL
LIN {X 0,Y 334.118,Z 398.867,A -85,B 0,C 180,E1 -14402.411,E2 -14402.411} C_VEL
LIN {X 0,Y 334.005,Z 398.877,A -85,B 0,C 180,E1 -14407.253,E2 -14407.253} C_VEL
LIN {X 0,Y 333.817,Z 398.904,A -85,B 0,C 180,E1 -14410.923,E2 -14410.923} C_VEL
LIN {X 0,Y 333.787,Z 398.907,A -85,B 0,C 180,E1 -14414.636,E2 -14414.636} C_VEL
LIN {X 0,Y 333.777,Z 398.903,A -85,B 0,C 180,E1 -14418.658,E2 -14418.658} C_VEL
LIN {X 0,Y 333.676,Z 398.92,A -85,B 0,C 180,E1 -14422.28,E2 -14422.28} C_VEL
LIN {X 0,Y 333.718,Z 398.914,A -85,B 0,C 180,E1 -14426.248,E2 -14426.248} C_VEL
LIN {X 0,Y 333.693,Z 398.917,A -85,B 0,C 180,E1 -14428.974,E2 -14428.974} C_VEL
LIN {X 0,Y 333.626,Z 398.923,A -85,B 0,C 180,E1 -14432.589,E2 -14432.589} C_VEL
LIN {X 0,Y 333.66,Z 398.924,A -85,B 0,C 180,E1 -14436.141,E2 -14436.141} C_VEL
LIN {X 0,Y 333.669,Z 398.923,A -85,B 0,C 180,E1 -14439.19,E2 -14439.19} C_VEL
LIN {X 0,Y 333.689,Z 398.922,A -85,B 0,C 180,E1 -14442.516,E2 -14442.516} C_VEL
LIN {X 0,Y 333.769,Z 399.103,A -85,B 0,C 180,E1 -14445.719,E2 -14445.719} C_VEL
LIN {X 0,Y 334.878,Z 404.696,A -85,B 0,C 180,E1 -14449.419,E2 -14449.419} C_VEL
LIN {X 0,Y 335.885,Z 410.149,A -85,B 0,C 180,E1 -14452.666,E2 -14452.666} C_VEL
LIN {X 0,Y 337.024,Z 415.623,A -85,B 0,C 180,E1 -14455.738,E2 -14455.738} C_VEL
LIN {X 0,Y 337.615,Z 419.919,A -85,B 0,C 180,E1 -14457.944,E2 -14457.944} C_VEL
LIN {X 0,Y 337.003,Z 424.194,A -85,B 0,C 180,E1 -14459.97,E2 -14459.97} C_VEL
LIN {X 0,Y 335.421,Z 433.875,A -85,B 0,C 180,E1 -14464.287,E2 -14464.287} C_VEL
LIN {X 0,Y 334.34,Z 441.957,A -85,B 0,C 180,E1 -14467.771,E2 -14467.771} C_VEL
LIN {X 0,Y 334.146,Z 443.742,A -85,B 0,C 180,E1 -14468.528,E2 -14468.528} C_VEL
LIN {X 0,Y 336.775,Z 457.163,A -85,B 0,C 180,E1 -14469.224,E2 -14469.224} C_VEL
LIN {X 0,Y 338.242,Z 469.319,A -85,B 0,C 180,E1 -14470.036,E2 -14470.036} C_VEL
LIN {X 0,Y 338.878,Z 480.296,A -85,B 0,C 180,E1 -14470.938,E2 -14470.938} C_VEL
LIN {X 0,Y 338.478,Z 486.894,A -85,B 0,C 180,E1 -14471.543,E2 -14471.543} C_VEL
LIN {X 0,Y 337.139,Z 497.732,A -85,B 0,C 180,E1 -14472.722,E2 -14472.722} C_VEL
LIN {X 0,Y 335.748,Z 508.49,A -85,B 0,C 180,E1 -14474.213,E2 -14474.213} C_VEL
LIN {X 0,Y 334.733,Z 517.194,A -85,B 0,C 180,E1 -14475.721,E2 -14475.721} C_VEL
LIN {X 0,Y 333.75,Z 525.584,A -85,B 0,C 180,E1 -14477.538,E2 -14477.538} C_VEL
LIN {X 0,Y 332.99,Z 531.305,A -85,B 0,C 180,E1 -14479.053,E2 -14479.053} C_VEL
LIN {X 0,Y 332.377,Z 539.229,A -85,B 0,C 180,E1 -14481.491,E2 -14481.491} C_VEL
LIN {X 0,Y 332.102,Z 543.898,A -85,B 0,C 180,E1 -14483.319,E2 -14483.319} C_VEL
LIN {X 0,Y 331.996,Z 547.412,A -85,B 0,C 180,E1 -14485.145,E2 -14485.145} C_VEL
LIN {X 0,Y 332.014,Z 549.149,A -85,B 0,C 180,E1 -14486.362,E2 -14486.362} C_VEL
LIN {X 0,Y 331.965,Z 550.451,A -85,B 0,C 180,E1 -14487.576,E2 -14487.576} C_VEL
LIN {X 0,Y 331.992,Z 551.345,A -85,B 0,C 180,E1 -14488.79,E2 -14488.79} C_VEL
LIN {X 0,Y 332.006,Z 551.798,A -85,B 0,C 180,E1 -14490.003,E2 -14490.003} C_VEL
LIN {X 0,Y 331.979,Z 551.815,A -85,B 0,C 180,E1 -14491.216,E2 -14491.216} C_VEL
LIN {X 0,Y 331.967,Z 551.433,A -85,B 0,C 180,E1 -14492.429,E2 -14492.429} C_VEL
LIN {X 0,Y 332.014,Z 550.649,A -85,B 0,C 180,E1 -14493.644,E2 -14493.644} C_VEL
LIN {X 0,Y 332.014,Z 548.184,A -85,B 0,C 180,E1 -14495.793,E2 -14495.793} C_VEL
LIN {X 0,Y 332.358,Z 544.446,A -85,B 0,C 180,E1 -14497.903,E2 -14497.903} C_VEL
LIN {X 0,Y 332.816,Z 540.059,A -85,B 0,C 180,E1 -14499.728,E2 -14499.728} C_VEL
LIN {X 0,Y 333.506,Z 534.473,A -85,B 0,C 180,E1 -14501.551,E2 -14501.551} C_VEL
LIN {X 0,Y 334.583,Z 527.526,A -85,B 0,C 180,E1 -14503.362,E2 -14503.362} C_VEL
LIN {X 0,Y 335.859,Z 518.867,A -85,B 0,C 180,E1 -14505.165,E2 -14505.165} C_VEL
LIN {X 0,Y 337.041,Z 510.292,A -85,B 0,C 180,E1 -14506.633,E2 -14506.633} C_VEL
LIN {X 0,Y 338.629,Z 499.4,A -85,B 0,C 180,E1 -14508.141,E2 -14508.141} C_VEL
LIN {X 0,Y 340.331,Z 487.236,A -85,B 0,C 180,E1 -14509.453,E2 -14509.453} C_VEL
LIN {X 0,Y 340.769,Z 480.823,A -85,B 0,C 180,E1 -14510.054,E2 -14510.054} C_VEL
LIN {X 0,Y 340.196,Z 469.422,A -85,B 0,C 180,E1 -14511.032,E2 -14511.032} C_VEL
LIN {X 0,Y 338.244,Z 455.159,A -85,B 0,C 180,E1 -14512.08,E2 -14512.08} C_VEL
LIN {X 0,Y 335.103,Z 441.135,A -85,B 0,C 180,E1 -14512.949,E2 -14512.949} C_VEL
LIN {X 0,Y 334.429,Z 437.976,A -85,B 0,C 180,E1 -14513.144,E2 -14513.144} C_VEL
LIN {X 0,Y 335.73,Z 427.865,A -85,B 0,C 180,E1 -14517.424,E2 -14517.424} C_VEL
LIN {X 0,Y 336.921,Z 420.402,A -85,B 0,C 180,E1 -14520.656,E2 -14520.656} C_VEL
LIN {X 0,Y 337.113,Z 417.156,A -85,B 0,C 180,E1 -14522.117,E2 -14522.117} C_VEL
LIN {X 0,Y 335.918,Z 410.527,A -85,B 0,C 180,E1 -14525.318,E2 -14525.318} C_VEL
LIN {X 0,Y 334.507,Z 403.215,A -85,B 0,C 180,E1 -14529.075,E2 -14529.075} C_VEL
LIN {X 0,Y 333.664,Z 398.925,A -85,B 0,C 180,E1 -14531.468,E2 -14531.468} C_VEL
LIN {X 0,Y 333.597,Z 398.931,A -85,B 0,C 180,E1 -14534.25,E2 -14534.25} C_VEL
LIN {X 0,Y 333.644,Z 398.926,A -85,B 0,C 180,E1 -14537.618,E2 -14537.618} C_VEL
LIN {X 0,Y 333.642,Z 398.921,A -85,B 0,C 180,E1 -14541.207,E2 -14541.207} C_VEL
LIN {X 0,Y 333.683,Z 398.92,A -85,B 0,C 180,E1 -14543.861,E2 -14543.861} C_VEL
LIN {X 0,Y 333.652,Z 398.923,A -85,B 0,C 180,E1 -14547.414,E2 -14547.414} C_VEL
LIN {X 0,Y 333.657,Z 398.924,A -85,B 0,C 180,E1 -14551.022,E2 -14551.022} C_VEL
LIN {X 0,Y 333.67,Z 398.923,A -85,B 0,C 180,E1 -14555.086,E2 -14555.086} C_VEL
LIN {X 0,Y 333.673,Z 398.923,A -85,B 0,C 180,E1 -14559.018,E2 -14559.018} C_VEL
LIN {X 0,Y 333.802,Z 398.907,A -85,B 0,C 180,E1 -14561.589,E2 -14561.589} C_VEL
LIN {X 0,Y 333.817,Z 398.906,A -85,B 0,C 180,E1 -14565.577,E2 -14565.577} C_VEL
LIN {X 0,Y 333.822,Z 398.904,A -85,B 0,C 180,E1 -14569.077,E2 -14569.077} C_VEL
LIN {X 0,Y 333.863,Z 399.019,A -85,B 0,C 180,E1 -14570.381,E2 -14570.381} C_VEL
LIN {X 0,Y 334.67,Z 402.683,A -85,B 0,C 180,E1 -14572.761,E2 -14572.761} C_VEL
LIN {X 0,Y 335.215,Z 406.553,A -85,B 0,C 180,E1 -14575.189,E2 -14575.189} C_VEL
LIN {X 0,Y 335.248,Z 410.701,A -85,B 0,C 180,E1 -14577.597,E2 -14577.597} C_VEL
LIN {X 0,Y 334.732,Z 416.036,A -85,B 0,C 180,E1 -14580.601,E2 -14580.601} C_VEL
LIN {X 0,Y 334.226,Z 423.499,A -85,B 0,C 180,E1 -14584.824,E2 -14584.824} C_VEL
LIN {X 0,Y 333.962,Z 428.916,A -85,B 0,C 180,E1 -14587.832,E2 -14587.832} C_VEL
LIN {X 0,Y 338.32,Z 442.883,A -85,B 0,C 180,E1 -14588.921,E2 -14588.921} C_VEL
LIN {X 0,Y 340.82,Z 453.813,A -85,B 0,C 180,E1 -14589.874,E2 -14589.874} C_VEL
LIN {X 0,Y 342.214,Z 463.412,A -85,B 0,C 180,E1 -14590.801,E2 -14590.801} C_VEL
LIN {X 0,Y 340.88,Z 475.023,A -85,B 0,C 180,E1 -14591.898,E2 -14591.898} C_VEL
LIN {X 0,Y 339.348,Z 486.25,A -85,B 0,C 180,E1 -14593.243,E2 -14593.243} C_VEL
LIN {X 0,Y 337.793,Z 496.49,A -85,B 0,C 180,E1 -14594.765,E2 -14594.765} C_VEL
LIN {X 0,Y 336.28,Z 505.829,A -85,B 0,C 180,E1 -14596.513,E2 -14596.513} C_VEL
LIN {X 0,Y 335.034,Z 513.658,A -85,B 0,C 180,E1 -14598.34,E2 -14598.34} C_VEL
LIN {X 0,Y 333.954,Z 520.36,A -85,B 0,C 180,E1 -14600.318,E2 -14600.318} C_VEL
LIN {X 0,Y 333.064,Z 525.608,A -85,B 0,C 180,E1 -14602.322,E2 -14602.322} C_VEL
LIN {X 0,Y 332.671,Z 528.388,A -85,B 0,C 180,E1 -14603.665,E2 -14603.665} C_VEL
LIN {X 0,Y 332.422,Z 530.562,A -85,B 0,C 180,E1 -14605.013,E2 -14605.013} C_VEL
LIN {X 0,Y 331.969,Z 533.049,A -85,B 0,C 180,E1 -14607.228,E2 -14607.228} C_VEL
LIN {X 0,Y 331.729,Z 534.17,A -85,B 0,C 180,E1 -14609.698,E2 -14609.698} C_VEL
LIN {X 0,Y 331.678,Z 533.703,A -85,B 0,C 180,E1 -14612.049,E2 -14612.049} C_VEL
LIN {X 0,Y 331.795,Z 531.783,A -85,B 0,C 180,E1 -14614.298,E2 -14614.298} C_VEL
LIN {X 0,Y 332.156,Z 528.528,A -85,B 0,C 180,E1 -14616.481,E2 -14616.481} C_VEL
LIN {X 0,Y 332.549,Z 524.061,A -85,B 0,C 180,E1 -14618.558,E2 -14618.558} C_VEL
LIN {X 0,Y 333.059,Z 518.259,A -85,B 0,C 180,E1 -14620.564,E2 -14620.564} C_VEL
LIN {X 0,Y 333.793,Z 511.007,A -85,B 0,C 180,E1 -14622.527,E2 -14622.527} C_VEL
LIN {X 0,Y 334.566,Z 503.436,A -85,B 0,C 180,E1 -14624.176,E2 -14624.176} C_VEL
LIN {X 0,Y 335.675,Z 493.652,A -85,B 0,C 180,E1 -14625.887,E2 -14625.887} C_VEL
LIN {X 0,Y 336.723,Z 483.202,A -85,B 0,C 180,E1 -14627.368,E2 -14627.368} C_VEL
LIN {X 0,Y 337.727,Z 473.126,A -85,B 0,C 180,E1 -14628.516,E2 -14628.516} C_VEL
LIN {X 0,Y 338.794,Z 460.146,A -85,B 0,C 180,E1 -14629.685,E2 -14629.685} C_VEL
LIN {X 0,Y 337.121,Z 448.646,A -85,B 0,C 180,E1 -14630.59,E2 -14630.59} C_VEL
LIN {X 0,Y 334.369,Z 434.52,A -85,B 0,C 180,E1 -14631.457,E2 -14631.457} C_VEL
LIN {X 0,Y 332.948,Z 427.622,A -85,B 0,C 180,E1 -14631.8,E2 -14631.8} C_VEL
LIN {X 0,Y 333.251,Z 421.199,A -85,B 0,C 180,E1 -14635.333,E2 -14635.333} C_VEL
LIN {X 0,Y 333.535,Z 414.706,A -85,B 0,C 180,E1 -14638.917,E2 -14638.917} C_VEL
LIN {X 0,Y 333.789,Z 408.416,A -85,B 0,C 180,E1 -14642.403,E2 -14642.403} C_VEL
LIN {X 0,Y 334.072,Z 402.369,A -85,B 0,C 180,E1 -14645.778,E2 -14645.778} C_VEL
LIN {X 0,Y 333.821,Z 398.905,A -85,B 0,C 180,E1 -14647.803,E2 -14647.803} C_VEL
LIN {X 0,Y 333.796,Z 398.908,A -85,B 0,C 180,E1 -14651.587,E2 -14651.587} C_VEL
LIN {X 0,Y 333.81,Z 398.905,A -85,B 0,C 180,E1 -14655.574,E2 -14655.574} C_VEL
LIN {X 0,Y 333.834,Z 398.902,A -85,B 0,C 180,E1 -14659.076,E2 -14659.076} C_VEL
LIN {X 0,Y 333.968,Z 398.886,A -85,B 0,C 180,E1 -14662.744,E2 -14662.744} C_VEL
LIN {X 0,Y 333.786,Z 398.913,A -85,B 0,C 180,E1 -14665.166,E2 -14665.166} C_VEL
LIN {X 0,Y 333.899,Z 398.94,A -85,B 0,C 180,E1 -14666.981,E2 -14666.981} C_VEL
